(* CODESYS project aircomlib_v1_3_0.library
   Author: Piotr Kaźmierczuk
   Placeholder: AircomLibrary
   Title: AircomLibrary
   Version: 1.3.0
   Description: Biblioteka z używanymi na liniach produkcyjnych oraz maszynach testowych blokami funkcyjnymi, strukturami danych,wizualizacjami etc.
   Company: AirCom

Project tree, tasks and I/O mapping:
  libraries: Tc2_Math, * (Beckhoff Automation GmbH); Tc2_SerialCom, * (Beckhoff Automation GmbH); Tc2_Standard, * (Beckhoff Automation GmbH); Tc2_System, * (Beckhoff Automation GmbH); Tc2_Utilities, * (Beckhoff Automation GmbH); Tc3_Database, * (Beckhoff Automation GmbH); Tc3_EventLogger, * (Beckhoff Automation GmbH); Tc3_Module, * (Beckhoff Automation GmbH); Util, * (System); VisuDialogs, * (System); VisuSymbols, * (System)
  Common/
    2HandStart/
      BasicVer/
        function block fb2HandStartBasic [ST]
        data type st2HandStartBasic_InOuts
      function block fb2HandStart [ST]
      data type st2HandStart_InOuts
    Actuator/
      function block fbActuator [ST]: mClose, mOpen, mReset, mStop
      function block fbActuatorOOP [ST]: ACT_Stop, mClose, mOpen, mReset, mStop
      function block fbActuatorV2 [ST]: mClose, mOpen, mReset, mStop, Closed, CmdsCounter, Moving, Opened
      data type stActuatorDigInOut
      data type stActuatorInOuts
    AlarmTable/
      DUTs/
        data type enAlarmClasses
        data type stAlarmRowAppearanceData
        data type stAlarmTableRow
      function f_AlarmClassToUINT [ST]
      function f_AlarmEnableTest [ST]
      function block fbAlarmMasterTable [ST]: mPopRows, mPushRow, mReset
      function block fbAlarmSlaveTable [ST]: aMesagesPoped, mPushRow, mReset
    LoadCell/
      function fLoadCellCtrl [ST]
      function fLoadCellStatusToBOOL [ST]
      data type stLoadCell_InOutsData
    Maintenance/
      function block fbIIS_Restart [ST]
      function block fbTcAdsWcfHost_Restart [ST]
    Measurement_Analog/
      function fACRoundReal [ST]
      function block FB_FilterEx [ST]
      function block fbAnalogMeasurement [ST]
      function block fbAnalogMonitor [ST]
      function fMeanFilter [ST]
      function fMeasureStatusToBOOL [ST]
      function fRealValueFilter [ST]
      data type stMeasurementScalingData
    PulseCounter/
      function block fbPulseCounter [ST]
      function block fbPulseCounterPIM [ST]
    RecipeManager/
      DUTs/
        data type nRecipeManager_ErrorList
        data type stRecipeManager_ListEntry
      VISUs/
        visualisation vRecipeManager_Ctrl
        visualisation vRecipeManager_CtrlWide
      function block fbRecipeManager [ST]: ACT_DeleteRecipe, ACT_ReadRecipe, ACT_RefreshRecipeList, ACT_WriteRecipe
    SerialCom/
      function block fbSerialLinkCommunication [ST]
      data type stSerialComData
    String Functions/
      function block fbAcFormatString [ST]
      function block fbConcatStrings [ST]
      function fDataToHexStr [ST]
      function fGetStringUntil [ST]
      function fHexStrToData [ST]
      function fRemChar [ST]
    TimeProg/
      function block fbDateAndTimeCalc [ST]: mCalculate
      data type stAircomTimeStruct
    TimeTableStats/
      OOP_Version/
        function block fbTimeTable255 [ST]: mPushRow, mPushText, mReset, IsEmpty, IsFull, LastIndex
        interface I_TimeTable255: mPushRow, mPushText, mReset, IsEmpty, IsFull, LastIndex
        data type stTimeStatsRow255
      function block fbTimeTable [ST]: mPushRow, mPushText, mReset, IsEmpty, IsFull, LastIndex, MaxIndex
      interface I_TimeTable: mPushRow, mPushText, mReset, IsEmpty, IsFull, LastIndex, MaxIndex
      data type stTimeStatsRow
    function block fbBinaryFilter [ST]
    function block fbBlink [ST]
    function block fbLED_Blink [ST]
    function block fbOperationSynch [ST]
    function block fbPwmGenerator [ST]
    function block fbSequenceWork [ST]
    function block fbWriteStringToFile [ST]
  DataLoggers/
    function block fbTextDataLogger [ST]: mAddLine, mAppendCurrentLine, mEndLine, mIsActEmpty, mSaveBuffor
  DUTs/
    data type nBasicWorkStep
  PIM/
    DUTs/
      data type nPIM_ErrorCodes
      data type nPIM_EventClasses
      data type nPIM_MachineStates
      data type nPIM_ReportedNokSource
      data type nPIM_ReworkSelect
      data type stPIM_ExtDataRow
      data type stPIM_MachineParametersData
      data type stPIM_ServiceInOuts
      data type stPIM_StationSettings
      data type stPIM_StationStatus
    Interfaces/
      interface I_PIM: m_SqlInsertExtendedData, m_SqlSelLastOperationStatus, mGetStationData, mNewEvent, mNewServiceMessage, mSetNewMachineState, PartsCtr_NOK, PartsCtr_OK, prActiveErrorCode, prCMD, prCurrentMachineState, prErrorClassExt, prErrorConfirmActive, prExternalEvtWaitInQueue, prLastSavedStatus, prNokReportedSource, prOperEnded, prOperInProgress, prPimActive, prPimBlockWork, prPlcBlockWork, prReworkStatus, prStationDataOK, prTestMode, prUserLogged, prWorkPermission, prIsEol, prPartCodeNumber, prIsHidden, prLineName, prMachNumber, prStationAlias, prStationName
      interface I_SqlCmds: m_SqlInsAdditionalError, m_SqlInsCompressedAirConsumption, m_SqlInsDefectRelation, m_SqlInsEnergyConsumption, m_SqlInsertExtendedData, m_SqlSelInsStatus, m_SqlSelLastOperationStatus
      interface I_StationMachine: mGetParamsData
    POUs/
      function block fbPIM_Dummy [ST]: m_SqlInsertExtendedData, m_SqlSelLastOperationStatus, mGetStationData, mNewEvent, mNewServiceMessage, mSetNewMachineState
      function block fbPIM_MachineDummy [ST]: FB_init, mGetParamsData, mNewEvent
      function block fbPIM_SimplePimStation [ST]: PartsCtr_NOK, PartsCtr_OK, prActiveErrorCode, prCMD, prCurrentMachineState, prErrorClassExt, prErrorConfirmActive, prExternalEvtWaitInQueue, prLastSavedStatus, prNokReportedSource, prOperEnded, prOperInProgress, prPimActive, prPimBlockWork, prPlcBlockWork, prReworkStatus, prStationDataOK, prTestMode, prUserLogged, prWorkPermission, prIsEol, prPartCodeNumber, prIsHidden, prLineName, prMachNumber, prStationAlias, prStationName, m_SqlInsAdditionalError, m_SqlInsCompressedAirConsumption, m_SqlInsDefectRelation, m_SqlInsEnergyConsumption, m_SqlInsertExtendedData, m_SqlInsMachineParamsData, m_SqlSelInsStatus, m_SqlSelLastOperationStatus, m_SqlSelLineStationId, m_SqlSelMachineParamsCRC, m_SqlSelMachineParamsData, ACT_PimCmdsHandling, ACT_SqlDataReturnCmd, ACT_UpdatePimOutput, FB_init, mGetStationData, mNewEvent, mSendCmdToPIM
      function block fbPIM_Station_V3 [ST]: PartsCtr_NOK, PartsCtr_OK, prActiveErrorCode, prCMD, prCurrentMachineState, prErrorClassExt, prErrorConfirmActive, prExternalEvtWaitInQueue, prLastSavedStatus, prNokReportedSource, prOperEnded, prOperInProgress, prPimActive, prPimBlockWork, prPlcBlockWork, prReworkStatus, prStationDataOK, prTestMode, prUserLogged, prWorkPermission, prIsEol, prPartCodeNumber, prIsHidden, prLineName, prMachNumber, prStationAlias, prStationName, m_SqlInsAdditionalError, m_SqlInsCompressedAirConsumption, m_SqlInsDefectRelation, m_SqlInsEnergyConsumption, m_SqlInsertExtendedData, m_SqlInsMachineParamsData, m_SqlSelInsStatus, m_SqlSelLastOperationStatus, m_SqlSelLineStationId, m_SqlSelMachineParamsCRC, m_SqlSelMachineParamsData, ACT_PimCmdsHandling, ACT_SqlDataReturnCmd, ACT_UpdatePimOutput, FB_init, mGetStationData, mNewEvent, mNewEventCommon, mNewlnternalEvent, mNewServiceMessage, mSendCmdToPIM, mSetNewMachineState
      function block fbPIM_UserLogin [ST]: FB_init
      function fPIM_GetCmdPar [ST]
  ProdLineMachines/
    AssemblyPost/
      DUTs/
        data type nAssemblyPost_ErrorList
        data type stAssemblyPost_Settings
      VISUs/
        visualisation vAssemblyPost_Main
      function block fbAssemblyPost [ST]: FB_init, mGetParamsData, mNewEvent
    S02_ManometerTubeAssy/
      V1/
        DUTs/
          data type nManometerTubeAssy_ErrorCodes
          data type stManometerTubeAssy_InOuts
        function block fbManometerTubeAssy_V1 [ST]: FB_init, mGetParamsData, mNewEvent
      V2/
        DUTs/
          data type nManometerTubeAssy_V2_ErrorCodes
          data type stManometerTubeAssy_V2_InOuts
        function block fbManometerTubeAssy_V2 [ST]: FB_init, mGetParamsData, mNewEvent
    S05_BallsWheelPress/
      DUTs/
        data type nBallCounterPressPress_ErrorCodes
        data type stBallCounterWeightPress_InOuts
        data type stBallCounterWeightPress_Params
      function block fbBallCounterWeightPress [ST]: FB_init, mGetParamsData, mNewEvent
    S11_ResWelderTecna/
      DUTs/
        data type nTecnaResWelder_ErrorCodes
        data type stTecnaResWelder_InOuts
        data type stTecnaResWelder_TestParams
      function block fbTecnaResWelder [ST]: FB_init, mGetParamsData, mNewEvent
    S12_Hios/
      DUTs/
        data type nHIOS_ErrorList
        data type nHIOS_SerialCmds
        data type stHIOS_FastenExtData
        data type stHIOS_InOuts
        data type stHIOS_ScrewDriverParams
        data type stHIOS_TestParameters
      function block fbHIOS_ScrewDriver [ST]: ACT_SerialCom, FB_init, mGetParamsData, mNewEvent
    S13_FrontFanPress/
      DUTs/
        data type nFrontFanPress_ErrorCodes
        data type stFrontFanPress_InOuts
      function block fbFrontFanPress [ST]: FB_init, mGetParamsData, mNewEvent
    S18_ManometerCalib/
      DUTs/
        data type nManometerCalibration_ErrorCodes
        data type stManometerCalibration_InOuts
        data type stManometerCalibration_TestData
      function block fbManometerCalibration [ST]: FB_init, mGetParamsData, mNewEvent
    Sonictech/
      Fixtures/
        NoWeldLock/
          function block fbStFix_NoWeldLock [ST]
          data type nStFix_NoWeldLock_ErrorCodes
        S01_IndicatorAssembly/
          DUTs/
            data type nStFix_S01IndicatorAssy_ErrorCodes
            data type stStFix_S01IndicatorAssy_InOut
            data type stStFix_S01IndicatorAssy_Settings
          VISUs/
            SubFrame/
              visualisation vStFix_S01IndicatorAssy_SubDiag
              visualisation vStFix_S01IndicatorAssy_SubSettings
            visualisation vStFix_S01IndicatorAssy_Main
          function block fbStFix_S01IndicatorAssy [ST]
        S06_CarrierWheelLubrification/
          V1/
            DUTs/
              data type nStFix_S06CarrierAndWheelAssyGrease_ErrorCodes
              data type stStFix_S06CarrierAndWheelAssyGrease_InOuts
              data type stStFix_S06CarrierAndWheelAssyGrease_Settings
            function block fbStFix_S06CarrierAndWheelAssyGrease [ST]
          V2/
            DUTs/
              data type nStFix_S06CarrierAndWheelAssyGrease_V2_ErrorCodes
              data type stStFix_S06CarrierAndWheelAssyGrease_V2_InOuts
              data type stStFix_S06CarrierAndWheelAssyGrease_V2_Settings
            function block fbStFix_S06CarrierAndWheelAssyGrease_V2 [ST]
        S07_CarrierAssyWithPiston/
          V1/
            DUTs/
              data type nStFix_S07CarrierPistonAssy_ErrorCodes
              data type stStFix_S07CarrierPistonAssy_InOuts
              data type stStFix_S07CarrierPistonAssy_Settings
            function block fbStFix_S07CarrierPistonAssy [ST]
          V2/
            DUTs/
              data type nStFix_S07CarrierPistonAssy_V2_ErrorCodes
              data type stMachineSettingsHeatStamp
              data type stStFix_S07CarrierPistonAssy_V2_InOuts
              data type stStFix_S07CarrierPistonAssy_V2_Settings
            function block fbStFix_S07CarrierPistonAssy_V2 [ST]: ACT_HeatStamp, mNewEvent
        S08_CoolerClosure/
          V1/
            function block fbStFix_S08CoolerClosure [ST]
            data type nStFix_S08CoolerClosure_ErrorCodes
            data type stStFix_S08CoolerClosure_InOuts
          V2/
            DUTs/
              data type nStFix_S08CoolerClosure_V2_ErrorCodes
              data type stStFix_S08CoolerClosure_V2_InOuts
              data type stStFix_S08CoolerClosure_V2_Settings
            function block fbStFix_S08CoolerClosure_V2 [ST]
        S10_CoolerCarrierOrifice/
          function block fbStFix_S10CoolerCarrierOrifice [ST]
          data type stStFix_S10CoolerCarrierOrifice_InOuts
        S16_FixAndFrontFanDetection/
          DUTs/
            data type nStFix_S16PinWeldFfDetection_ErrorCodes
            data type stStFix_S16PinWeldFfDetection_InOuts
            data type stStFix_S16PinWeldFfDetection_Settings
          function block fbStFix_S16PinWeldFfDetection [ST]
        S17_EnclosurePressFix/
          DUTs/
            data type nStFix_S17EnclosureWelding_ErrorCodes
            data type stStFix_S17EnclosureWelding_InOuts
          function block fbStFix_S17EnclosureWelding [ST]
        function block fbStFixBaseTemplate [ST]: prFixError, prFixErrorID, prFixLocked, prFixReady, prFixReleased, prMachState, prTestMode, prTestOutputsActive, prUserLogged, prWeldingActive, actCheckForNewOrder, mAuxOper, mLock, mNewEvent, mRelease
        interface I_Fixture: prFixError, prFixErrorID, prFixLocked, prFixReady, prFixReleased, prMachState, prTestMode, prTestOutputsActive, prUserLogged, prWeldingActive, mAuxOper, mLock, mRelease
      SerialCom/
        DUTs/
          DataStruct/
            data type stSonicTech_SerialStructGenParamsRange
            data type stSonicTech_SerialStructProgParams
            data type stSonicTech_SerialStructSoftVer
            data type stSonicTech_SerialStructWeldParams
          data type nSonicTech_SerialCmdClasses
          data type nSonicTech_SerialCmdStatus
          data type nSonicTech_SerialCmdType
          data type stSonicTech_SerialCMD
        function block fbSonictechSerialCom [ST]: ACT_Test_Cmds, mAddToQueue, mFillSendBuffor
        function block fbSonictechSerialRcv [ST]
        interface I_SonicTech_SerialCom: mAddToQueue
      Welding Machine/
        DUTs/
          data type nSonicTech_ErrorList
          data type stSonicTech_DigInOuts
          data type stSonicTech_MachSettings
        VISUs/
          SubFrame/
            visualisation vSonictechUSWM_SubDiag
            visualisation vSonictechUSWM_SubSettings
            visualisation vSonictechUSWM_SubStatus
          visualisation vSonictechUSWM_Main
        function block fbSonictechUSWM [ST]: FB_init, mGetParamsData, mNewEvent, mNewMachEvent
  SQL/
    DUTs/
      DataSelectDUTs/
        data type stSQL_RetDataProdLineStat
        data type stSQL_RetDataProdMachParams
        data type stSQL_RetDataUserRole
      HMI_DUTs/
        data type stSQL_HMI_CoreNodesData
        data type stSQL_HMI_QueueData
      data type nSQL_CmdExecState
      data type nSQL_CmdTypes
      data type nSQL_ErrorCodes
      data type nSQL_UserRoles
      data type stSQL_ClientNode
      data type stSQL_SaveStatustParams
    VISUs/
      visualisation vSQL_Core_AlarmTab
      visualisation vSQL_CoreDiag
    function block fbSQL_Core [ST]: actConnectionCheck, IsCoreWork, m_ErrorAnalysis, mAddCmdToQueue, mPopCmdFromQueue
    function block fbSQL_CoreNode [ST]: ACT_Init, mSaveError
    interface I_SQL_Core: IsCoreWork, mAddCmdToQueue
  VisionSensors/
    Balluff BVS/
      function block fbBvsControl [ST]: mNewInspection, mReadInspectionId, mSetInspectionId
      function block fbBvsControl_ComIO [ST]: mNewInspection, mReadInspectionId, mSetInspectionId
      data type stBVS_DigInOut
    Cognex/
      function block fbCognexIS280Control [ST]: mNewInspection, mReadInspectionId, mSetInspectionId
      data type stCognexIS280_DigInOut
    Keyence/
      IV3/
        data type stKeyenceIV3_DigInOut
      function block fbKeyenceIVControl [ST]: mNewInspection, mReadInspectionId, mSetInspectionId
      function block fbKeyenceIVControl_ComIO [ST]: mNewInspection, mReadInspectionId, mSetInspectionId
      data type stKeyence_DigInOut
    interface I_VisionSensorSTD: mNewInspection, mReadInspectionId, mSetInspectionId
    data type stVisionSensor_DigInOut
  text list GlobalTextList
  global variables GVL_Aircom
  program ReadMe [ST]
*)

// Common/2HandStart/BasicVer/st2HandStartBasic_InOuts
TYPE st2HandStartBasic_InOuts :
STRUCT
	bEmergButton_NC 	AT %I* :BOOL;		// TRUE- Emergency button released (inactive) , FALSE- Pressed (safety function activated)
	bLeftStart_NC 		AT %I* :BOOL;		// First button - NC contact
	bRightStart_NO 		AT %I* :BOOL;		// Second button - NO contact
END_STRUCT
END_TYPE

// Common/2HandStart/st2HandStart_InOuts
TYPE st2HandStart_InOuts :
STRUCT
	bSafetyStatus_NC 	AT %I* :BOOL;		// 1- gdy układ nie uzbrojony i sprawny (zezwolenie na reset), 0- gdy uzbrojony lub uszkodzony
	bEmergButton_NO 	AT %I* :BOOL;		// 1- Stop bezpieczeństwa wciśnięty, 0- zwolniony
	bLeftStart_NC 		AT %I* :BOOL;
	bRightStart_NO 		AT %I* :BOOL;
	bLeftStart_NO 		AT %I* :BOOL;
	bRightStart_NC 		AT %I* :BOOL;
	bSafetyReset 		AT %Q* :BOOL;		// Uzbrojenie układu bezpieczeństwa
END_STRUCT
END_TYPE

// Common/Actuator/stActuatorDigInOut
TYPE stActuatorDigInOut :
STRUCT
	bI_Opened AT %I*:BOOL;							// Sygnał z krańcówki otwarcia
	bI_Closed AT %I*:BOOL;							// Sygnał z krańcówki zamknięcia
	bQ_Open AT %Q*:BOOL:= FALSE;					// Sygnał do zaworu otwierania (w przypadku zaworu jednocewkowego podłączyć tylko to wyjście)
	bQ_Close AT %Q*:BOOL:= FALSE;					// Sygnał do zaworu zamykania
END_STRUCT
END_TYPE

// Common/Actuator/stActuatorInOuts
TYPE stActuatorInOuts :
STRUCT
	bI_Opened AT %I*:BOOL;							// Sygnał z krańcówki otwarcia
	bI_Closed AT %I*:BOOL;							// Sygnał z krańcówki zamknięcia
	bQ_Open AT %Q*:BOOL:= FALSE;					// Sygnał do zaworu otwierania (w przypadku zaworu jednocewkowego podłączyć tylko to wyjście)
	bQ_Close AT %Q*:BOOL:= FALSE;					// Sygnał do zaworu zamykania
END_STRUCT
END_TYPE

// Common/AlarmTable/DUTs/enAlarmClasses
{attribute 'qualified_only'}
{attribute 'strict'}
{attribute 'to_string'}
TYPE enAlarmClasses :
(
	// Lista klas alarmów - identyfikatory nie powinny zmieniać wartości
	None := 0,					// Logowanie wyłączone
	Info := 1,					// Logowanie podstawowych informacji
	Warning := 2,				// Ostrzeżenia
	Error := 4,	
	Quality := 8,
	Maintenance := 16,
	IT := 32,
	Developer := 64);
END_TYPE

// Common/AlarmTable/DUTs/stAlarmRowAppearanceData
TYPE stAlarmRowAppearanceData :
STRUCT
	sFontName:STRING:= 'Arial';
	iFontSize:INT:= 10;			// Rozmiar czcionki
	dwFontFlags:DWORD; 			// Flagi 1-italic, 2-bold, 4-underlined, 8-deleted, można je sumować
	dwTextColor:DWORD:=16#FF404040;			// Format koloru - 16#TTRRGGBB;
	dwAlignmentFlags:DWORD;		// Wyrównanie tekstu 0-TopLeft, 1-CenterHor, 2-Right, 4-CenterVert, 8-below
	dwBackgroundColor:DWORD:=16#FFCDCDCD;	// Kolor tła
	dwFrameColor:DWORD:=16#FF585858;		// Kolor ramki
	iFrameWidth:INT:= 1;					// Rozmiar ramki
END_STRUCT
END_TYPE

// Common/AlarmTable/DUTs/stAlarmTableRow
TYPE stAlarmTableRow :
STRUCT
	dtEventTime:DT;
	sMachineId:STRING(30);
	sEventDescription:STRING;
	dwErrorCode:DWORD;
	uiRepeatQty:UINT := 0;
	nAlarmClass:enAlarmClasses;
END_STRUCT
END_TYPE

// Common/LoadCell/stLoadCell_InOutsData
TYPE stLoadCell_InOutsData :
STRUCT
	wStatus		AT %I* : WORD;	// .1-Overrange, .3-Data invalid, .6-Error, .7-Calib in progress, .9-Steady state, .13-SyncErr, .15-TxPDO_Toggle
	rValue		AT %I* : REAL;	// Wartość siły w [N]
	wControl	AT %Q* : WORD;	// .0-Start calibration, .1-Disable calib., .2-InputFreeze, .4-Tara
END_STRUCT
END_TYPE

// Common/Measurement_Analog/stMeasurementScalingData
TYPE stMeasurementScalingData :
STRUCT
	rScalingRawValue_I:REAL := 0;	// Wartość surowa pomiaru w I punkcie pomiarowym
	rScalingEngValue_I:REAL	:= 0;		// Wartość inżynierska pomiaru w I punkcie pomiarowym
	rScalingRawValue_II:REAL := 32767;	// Wartość surowa pomiaru w II punkcie pomiarowym
	rScalingEngValue_II:REAL := 10;	// Wartość inżynierska pomiaru w II punkcie pomiarowym
END_STRUCT
END_TYPE

// Common/RecipeManager/DUTs/nRecipeManager_ErrorList
{attribute 'qualified_only'}
{attribute 'strict'}
{attribute 'to_string'}
TYPE nRecipeManager_ErrorList :
(
	NoError := 0,
	ReloadRecipeListError:= 1,
	WriteRecipeError := 2,
	ReadRecipeError := 3,
	WriteSizeError:= 4,
	ReadSizeError:= 5,
	StructToBig:= 6,
	FileOpenError:= 7,
	FileCloseError:= 8,
	ReadRecipeTimeout:= 9,
	WriteRecipeTimeout:= 10,
	BadCRC:= 11,
	CommandStartProgramError:=12,
	FileDeleteError:=13,
	DeleteRecipeTimeout := 14
);
END_TYPE

// Common/RecipeManager/DUTs/stRecipeManager_ListEntry
TYPE stRecipeManager_ListEntry :
STRUCT
	sFileName:STRING;
	dtCreationTime:DT;
END_STRUCT
END_TYPE

// Common/SerialCom/stSerialComData
TYPE stSerialComData :
STRUCT
	fbSerialCom			: fbSerialLinkCommunication;	// Blok odpowiedzialny za komunikacjię
	RxBufferEL			: ComBuffer;	// Receive data buffer; used with all receive function blocks *)
	TxBufferEL			: ComBuffer;	// Transmit data buffer; used with all receive function blocks 
END_STRUCT
END_TYPE

// Common/TimeProg/stAircomTimeStruct
TYPE stAircomTimeStruct :
STRUCT
	bTimeValid		: BOOL;					// Jeśli true dane w strukturze są aktualne
	stTimeStruct 	: TIMESTRUCT;			// Struktura z danymi rokiem, miesiącem, dniem itp w formacie WORD
	dtActualDate 	: DT;					// Aktualny czas typ DT
	tCycleTime		: TIME;					// Czas cyklu sterownika PLC
	tActualTime		: TIME;					// Aktualny czas
	sTimeString		: STRING(19);			// String z aktualną datą w formacie : YYYY-MM-DD hh:mm:ss
	sLogTimeString		: STRING(18);			// String z aktualną datą w formacie : MM-DD hh:mm:ss.uuu
	diPLC_UpTimeSeconds	: DINT:= 0;			// Licznik czasu pracy PLC w sekundach
	dtPLC_UpTime	: DT;					// Czas w którym PLC wystartował					
	// Znaczniki nowych okresów czasu
	bNew_Second_IMP, bNew_Minute_IMP, bNew_Hour_IMP, bNew_Day_IMP, bNew_Week_IMP, bNew_Month_IMP, bNew_Year_IMP:BOOL;	// Impuls nowej sekundy, minuty, godziny, dnia, tygodnia, miesiąca, roku
	// Znaczniki zmian
	bNew_Shift		: BOOL;					// Znacznik nowej zmiany (impuls)
	wWeekNb			: WORD;					// Numer tygodnia
	uiShiftNumber	: UINT;					// Numer aktualnej zmiany 1, 2 lub 3
END_STRUCT
END_TYPE

// Common/TimeTableStats/OOP_Version/stTimeStatsRow255
{attribute 'enable_dynamic_creation'}
TYPE stTimeStatsRow255 :
STRUCT
	sStepName:STRING(255);
	rStepTime:REAL;
END_STRUCT
END_TYPE

// Common/TimeTableStats/stTimeStatsRow
TYPE stTimeStatsRow :
STRUCT
	sStepName:STRING;
	rStepTime:REAL;
END_STRUCT
END_TYPE

// DUTs/nBasicWorkStep
{attribute 'qualified_only'}
{attribute 'strict'}
TYPE nBasicWorkStep :
(
	StartUpInicialization	 	:= 0,
	Inicialization			 	:= 5,
	WaitForStart	 			:=10,
	LockStation 				:=90,
	WaitForConfirm				:=94,
	ConfirmInProgress			:=95
);
END_TYPE

// PIM/DUTs/nPIM_ErrorCodes
{attribute 'qualified_only'}
{attribute 'strict'}
TYPE nPIM_ErrorCodes :
(
	// Common errors	
	NoError := 0,										// Brak błędu
	UnKnownAlarm := 53,									// Niezidentyfikowany alarm maszyny
	UnKnownLock := 54,									// Niezidentyfikowana blokada maszyny
	MachErrorWhenNoErrorCode := 56,						// Maszyna w oczekiwaniu na reset, ale brak błędu
	ProgramError := 90,									// Błąd w konfiguracji oprogramowania - zerowy wskaźńik itp
	SelectStationIdError := 230,						// Błąd pobrania ID stacji z bazy danych
	StatusSaveError := 89,								// Błąd zapisu statusu
	InputDependencyError := 99,							// Błąd zależności wejściowych (brak referencji)
	ResetTimeout := 518,								// Timeout resetu maszyny
	NoConfiguredOutPart := 150, 						// Brak skonfigurowanej części wyjściowej dla stanowiska
	NoMatchingParamsForComponent := 151,				// Brak zdefiniowanych parametrów dla komponentu
	ParamsMismatchPLCandDB := 152,						// Rozbieżność parametrów w PLC i w DB
	NoDbConnWorkAllowedTemporary := 153,				// Brak połączenia do DB, stacja dopuszczona warunkowo
	ParamsSaveToDB_Error := 154,						// Błąd wysłania parametrów programu do bazy danych
	ParamsReadFromDB_Error := 155,						// Błąd pobierania parametrów programu z bazy danych
	MachineParametersNoUpdated := 156					// Błąd odświeżenia danych z maszyny
);
END_TYPE

// PIM/DUTs/nPIM_EventClasses
{attribute 'qualified_only'}
{attribute 'to_string'}
{attribute 'strict'}
TYPE nPIM_EventClasses :
(
	NoError := 0,				// Brak błędu/alarmuwiadomości
	Message := 1,				// Wiadomość do użytkownika - baner wyświetlony przez x sekund lub do startu nowej operacji 
	AlarmAutoConfirm := 2,		// Alarm stanowiska który działa tak jak wprzypadku zwykłego alarmu ale zostaje automatycznie potwierdzony przy starcie nowej operacji 
	Alarm := 3,					// Alarm stanowiska - błąd związany z pracą maszyny, potwierdzenie nie wymaga lidera, nie ma pytania o rework
	Error := 4					// Blokowanie stanowiska powiązane z częścią - zawsze błąd potwierdza lider, sprawdzeny jest zapis statusu oraz część jest blokowana w kowadle (+ pytanie o rework)
);
END_TYPE

// PIM/DUTs/nPIM_MachineStates
{attribute 'qualified_only'}
{attribute 'strict'}
{attribute 'to_string'}
(*	Na podstawie stanu/kroków maszyny wydawane jest zezwolenie na przejście do danego kroku (zezwolenie na pracę, reset błędu itp) oraz zapisywany jest status operacji. 
	Wzorzec postępowania
	1. _2_ReadyForNewOperation - maszyna gotowa do wykonania operacji,
	2. _3_NewOperationStarted - gdy maszyna wystartowała blok stacji zapamiętuje konieczność zapisu statusu, 
	3. _5_OperationEndedOK lub _7_ErrorOccurr - informacja jaki status trzeba zapisać
	Jeśli po starcie operacji był sygnał _9_ErrorOccurr a nie było zapisu statusu (zgłoszenie błędu) i jest stan _10_WaitForReset to zapis statusu przez stację PIM

	Reset błędów: Blok maszyny czeka w stanie _8_WaitForReset zezwolenie na przejście do kolejnego kroku (_9_ResetInProgress). Jeśli reset zakończony powodzeniem zawsze kończy się stanem
	_0_Standby_NotReady (przy tym przejściu resetowane są zmienne od alarmów jeśli był aktywny błąd zewnętrzny)
*)
TYPE nPIM_MachineStates :
(
	_0_Initialization	 		:= 100,	// Inicjalizacja maszyny
	_0_Standby_NotReady 		:= 0,	// Maszyna w oczekiwaniu na stan gotowości
	_1_InManualControl		 	:= 1,	// Maszyna w sterowaniu serwisowym/ręcznym 
	_2_ReadyForNewOperation 	:= 2,	// Maszyna gotowa na wykonanie kolejnej operacji ( sygnał nie uwzględnia zezwolenia na pracę
	_3_NewOperationStarted 		:= 3,	// Nowa operacja rozpoczęta - jest zezwolenie, przygotowanie kowadła
	_4_OperationInProgress 		:= 4,	// Operacja w trakcie
	_5_OperationEndedOK			:= 5,	// Operacja zakończona ze statusem OK
	_6_ReturningToBaseState		:= 6,	// Powrót do stanu początkowego po zezwoleniu przez PIM
	_7_ErrorOccurr				:= 7,	// Wystąpił błąd - blokowanie części ustawianie maszyny w odpowiednim stanie	
	_8_WaitForReset				:= 8,	// Oczekiwanie na sygnał reset
	_9_ResetInProgress			:= 9	// Trwa reset maszyny
);
END_TYPE

// PIM/DUTs/nPIM_ReportedNokSource
{attribute 'qualified_only'}
{attribute 'strict'}
TYPE nPIM_ReportedNokSource :
(
	none := 0,
	FromPrevStation := 1,
	FromMach := 2,
	FromBox := 3,
	Error_UnknownSource := 4
);
END_TYPE

// PIM/DUTs/nPIM_ReworkSelect
{attribute 'qualified_only'}
{attribute 'strict'}
TYPE nPIM_ReworkSelect :
(
	none := 0,
	yes := 1,
	no := 2
);
END_TYPE

// PIM/DUTs/stPIM_ExtDataRow
TYPE stPIM_ExtDataRow :
STRUCT
	sName:STRING(63);		// Nazwa parametru
	sValue:STRING(31);		// Wartość parametru
END_STRUCT
END_TYPE

// PIM/DUTs/stPIM_MachineParametersData
TYPE stPIM_MachineParametersData :
STRUCT
	abMachineParameters: ARRAY [1..1000] OF BYTE;		// Wskaźnik do parametrów pracy maszyny
	uiMachineParametersSize: UINT;						// Rozmiar struktury parametrów pracy maszyny
	wActualCRC16SumInMachine: WORD;						// Aktualna suma CRC16 obliczona z parametrów
END_STRUCT
END_TYPE

// PIM/DUTs/stPIM_ServiceInOuts
(*
	Lista zmiennych które są wymieniane pomiędzy PLC a PIM, nazewnictwo zmiennych poszukiwanych w programie MAIN:
		stStacjaXXXX	- gdzie XXXX to nazwa stanowiska w PIM np. stStacjaLJ01, stStacjaLL19 - dla stanowisk z pojedynczą maszyną...
		stStacjaXXXX_MY	- gdzie XXXX to jw. nazwa stanowiska, Y to numer maszyny na stanowisku np. stStacjaLJ05_M1, stStacjaLJ05_M2 - dla stanowisk wielomaszynowych
	Update 01.03.2024r. - nowe nazwy zmiennych
		stStation_L{nazwa linii}_S{nazwa stanowiska}[_M{numer maszyny}] - rzeczy w klamrach {} zastępujemy zgodnie ze stanowiskiem, parametr z numerem maszyny w nawiasach [] jest konieczny tylko gdy maszyn jest >1
*)
TYPE stPIM_ServiceInOuts :
STRUCT
	//Dane in/out systemu PIM
	bPIMActive : BOOL := TRUE;					// jeśli TRUE system PIM wlaczony
	bUserLogged : BOOL := FALSE; 				// z PIM blokowanie stanowiska gdy nikt nie jest zalogowany - 1 nie zalogowany, 0 - zalogowany  
	bWorkBlock_PIM : BOOL;						// z PIM blokowane - 1 blokada, 0 praca
	bWorkBlock_PLC : BOOL;						// z PLC, jesli TRUE stanowisko pozostaje zablokowane z powodu błędu z operacją, trzeba wysłać status części NOK do bazy danych z kodem błędu
	bAlarmPLC : BOOL;							// z PLC, jesli TRUE stanowisko pozostaje zablokowane z powodu błędu maszyny, brak zapisu statusu (można zapisać dodatkowy kod błędu)
	bNonBlockingAlarm : BOOL;					// do użytku w kodzie PLC - gdy true i jest aktywny AlarmStanowiska, stanowisko nie jest blokowane (jedynie wyświetlany jest alarm - potwierdzenie po starcie nowej operacj, zniknięciu powodu błędu)
	bConfirmEvent : BOOL;						// z PIM potwierdzenie bledu, komunikatu przez operatora
	bTestMode : BOOL;							// jesli TRUE stacja nie sprawdza poprzedniej operacji 
	sErrorCodePLC : STRING(255); 				// komunikat o bledzie dzialania maszyny np kontaktron, e-stop
	sPlcServiceMessage : STRING(255);			// Komunikat do PIM wyświetlany na dolnym pasku
	sStatusNokAndErrorID : STRING(255);			// Informacja odczytywana przez PIM aby zapisać relację błędów - postaci {IdStatusu}:{IdBłędu}
	sCmdPIM2PLC:STRING(255);					// Komunikaty wysyłane z PIM do PLC (np. informacja o nowym boxie, zgłoszeniu części NOK itp)
	sCmdPLC2PIM:STRING(255);					// Komunikaty wysyłane z PLC do PIM  (np. zapytanie o licznik części itp.)
END_STRUCT
END_TYPE

// PIM/DUTs/stPIM_StationSettings
TYPE stPIM_StationSettings :
STRUCT
	bCheckMachineSettings:BOOL := FALSE;			// Sprawdzaj parametry maszyny
	bAutoRetooling:BOOL;							// Jeśli nastąpiło przezbrojenie automatycznie pobierz nowe parametry z bazy danych (o ile istnieją)
	bSkipCheckStatusSaveResult:BOOL:= FALSE;		// Czekaj z gotowością do nowej operacji aż status zostanie poprawnie zapisany
END_STRUCT
END_TYPE

// PIM/DUTs/stPIM_StationStatus
TYPE stPIM_StationStatus :
STRUCT
	// Dane informacyjne z bloczka obsługi PIM
	sLine				: STRING(31);	// Nazwa linii
	sStation			: STRING(31);	// Nazwa stacji
	sNazwaStanowiska 	: STRING(16);	// Id stanowiska (stanowisko + nr maszyny)
	
	stStationSqlData:stSQL_RetDataProdLineStat;	// Dane stanowiska - Id, AutSaveErrors itp	
	iMachineNumber 		: INT;			// Numer maszyny na stanowisku
	bIsHidden 			: BOOL;			// Czy ukrywanie zapisu statusu
	
			
(*	// Liczniki części oraz błędów
	iOutBoxQty, iOutBoxTargetQty: INT;			// liczba ilość części w pudełku wyjściowym - zmienne inkrementowane/dekrementowane tylko w bloczku PIM! Uaktualniane w FB maszyny tylko jeśli był restart sterownika.
	iPartsOK:INT;								// Licznik części OK wyprodukowanych na aktualnej zmianie
	iPartsNOK:INT;								// Licznik części NOK wyprodukowanych na aktualnej zmianie
	iPartsNotSaved:INT;							// Licznik błędnych statusów OK/NOK na aktualnej zmianie
	rEnergyConsumption:REAL;					// Zużycie energii na stanowisku	
	*)
END_STRUCT
END_TYPE

// ProdLineMachines/AssemblyPost/DUTs/nAssemblyPost_ErrorList
{attribute 'qualified_only'}
{attribute 'strict'}
TYPE nAssemblyPost_ErrorList :
(
	NoError := 0,
	PartRemovedToFast := 93,				// Złożenie zbyt szybko usunięte z kowadła
	PartInsertedToFast := 94,				// Złożenie zbyt szybko umieszczone w kowadle po usunięciu starego
	InputDependencyError := 99
);
END_TYPE

// ProdLineMachines/AssemblyPost/DUTs/stAssemblyPost_Settings
TYPE stAssemblyPost_Settings :
STRUCT
	bMonitorON_Time:BOOL;
	bMonitorOFF_Time:BOOL;
	rRequiredTimeON:REAL;
	rRequiredTimeOFF:REAL;
END_STRUCT
END_TYPE

// ProdLineMachines/S02_ManometerTubeAssy/V1/DUTs/nManometerTubeAssy_ErrorCodes
{attribute 'qualified_only'}
{attribute 'strict'}
{attribute 'to_string'}
TYPE nManometerTubeAssy_ErrorCodes :
(
	// Błędy ogólne
	NoError := 0,
	UnKnownAlarm := 53,						// Niezidentyfikowany alarm maszyny
	UnKnownLock := 54,						// Niezidentyfikowana blokada maszyny
	ProgramConfigError := 90,				// Błąd w konfiguracji programu
	ResetTimeout := 518,					// Timeout resetu maszyny
	SafetySystemNotArmed := 614,			// System safety nie uzbrojony
	NoMachineReactionOnStartSig := 140,		// Brak reakcji na sygnał startu (brak wysunięcia siłownika - brak powietrza itp.)
	TwoHandStartReleasedToEarly := 96,		// Dwustart zwolniony zbyt wcześnie
	
	TwoHandStartContactsError := 130,		// Błąd styków dwustartu
	WorkPosAchieveTimeout := 131,			// Nie osiągnięto pozycji roboczej w zadanym czasie
	OperInteruptedBeforeWorkPos := 132,		// Za wcześnie puszczono dwustart - część nie wprasowana
	WorkPosLost := 138,						// Utracona pozycja robocza (możliwy brak części)
	HomePosAchieveTimeout := 139			// Nie osiągnięto pozycji bazowej w zadanym czasie
//	InConsistentSignalsFromSensors := 1000	// Niewłaściwe odczyty stanów z czujników - ingerencja zewnętrzna 
);
END_TYPE

// ProdLineMachines/S02_ManometerTubeAssy/V1/DUTs/stManometerTubeAssy_InOuts
TYPE stManometerTubeAssy_InOuts :
STRUCT
	st2HandStartIO			: st2HandStartBasic_InOuts;	// Sygnały z układu dwu-startu
	bHandleWorkPos			AT %I*: BOOL;	
	bHandleHomePosV2		AT %I*: BOOL;	// USed only with V2 wersion
	bPressWorkPos			AT %I*: BOOL;	
	bPressHomePos			AT %I*: BOOL;	
	bPressValve_Q			AT %Q*: BOOL;	
END_STRUCT
END_TYPE

// ProdLineMachines/S02_ManometerTubeAssy/V2/DUTs/nManometerTubeAssy_V2_ErrorCodes
{attribute 'qualified_only'}
{attribute 'strict'}
{attribute 'to_string'}
TYPE nManometerTubeAssy_V2_ErrorCodes :
(
	// Błędy ogólne
	NoError := 0,
	UnKnownAlarm := 53,						// Niezidentyfikowany alarm maszyny
	UnKnownLock := 54,						// Niezidentyfikowana blokada maszyny
	ProgramConfigError := 90,				// Błąd w konfiguracji programu
	ResetTimeout := 518,					// Timeout resetu maszyny
	SafetySystemNotArmed := 614,			// System safety nie uzbrojony
	NoMachineReactionOnStartSig := 140,		// Brak reakcji na sygnał startu (brak wysunięcia siłownika - brak powietrza itp.)
	NoWorkPermittionFromPIM := 84,			// Brak zezwolenia na pracę
	TwoHandStartReleasedToEarly := 96,		// Dwustart zwolniony zbyt wcześnie
	PusherHomePositionError:= 120,			//Praska nie w pozycji bazowej
	PusherWorkPositionError:= 121,			//Praska nie w pozycji pracy
	CartridgeHomePositionError:= 122,		//Wózeczek nie w pozycji bazowej
	CartridgeWorkPositionError:= 123,		//Wózeczek nie w pozycji pracy
	WorkPosAchieveTimeout := 131,			// Nie osiągnięto pozycji roboczej w zadanym czasie
	OperInteruptedBeforeWorkPos := 132,		// Za wcześnie puszczono dwustart - część nie wprasowana
	WorkPosLost := 138,						// Utracona pozycja robocza (możliwy brak części)
	HomePosAchieveTimeout := 139,			// Nie osiągnięto pozycji bazowej w zadanym czasie
	OperationTooEarly	:= 182				// Operacja została wykonanna w zbyt krótkim czasie 
);
END_TYPE

// ProdLineMachines/S02_ManometerTubeAssy/V2/DUTs/stManometerTubeAssy_V2_InOuts
TYPE stManometerTubeAssy_V2_InOuts :
STRUCT
	st2HandStartIO			: st2HandStartBasic_InOuts;	// Sygnały z układu dwu-startu
	bMoverWorkPos			AT %I*: BOOL;	
	bPressWorkPos			AT %I*: BOOL;	
	bPressHomePos			AT %I*: BOOL;	
	bMoveValve_Q			AT %Q*: BOOL;
	bPressValve_Q			AT %Q*: BOOL;	
END_STRUCT
END_TYPE

// ProdLineMachines/S05_BallsWheelPress/DUTs/nBallCounterPressPress_ErrorCodes
{attribute 'qualified_only'}
{attribute 'strict'}
{attribute 'to_string'}
TYPE nBallCounterPressPress_ErrorCodes :
(
		// Błędy ogólne
	NoError := 0,
	UnKnownAlarm := 53,						// Niezidentyfikowany alarm maszyny
	UnKnownLock := 54,						// Niezidentyfikowana blokada maszyny
	ProgramConfigError := 90,				// Błąd w konfiguracji programu
	ResetTimeout := 518,					// Timeout resetu maszyny
	SafetySystemNotArmed := 614,			// System safety nie uzbrojony
	NoMachineReactionOnStartSig := 140,		// Brak reakcji na sygnał startu (brak wysunięcia siłownika - brak powietrza itp.)
	TwoHandStartReleasedToEarly := 96,		// Dwustart zwolniony zbyt wcześnie

	WorkPosAchieveTimeout := 131,			// Nie osiągnięto pozycji roboczej w zadanym czasie
	OperInteruptedBeforeWorkPos := 132,		// Za wcześnie puszczono dwustart - część nie wprasowana
	WorkPosLost := 138,						// Utracona pozycja robocza (możliwy brak części)
	HomePosAchieveTimeout := 139,			// Nie osiągnięto pozycji bazowej prasy w zadanym czasie
	BallsNotPresentAfterPushing := 142

);
END_TYPE

// ProdLineMachines/S05_BallsWheelPress/DUTs/stBallCounterWeightPress_InOuts
TYPE stBallCounterWeightPress_InOuts :
STRUCT
	bPressUpPosition		AT %I* :BOOL;
	bPressDownPosition		AT %I* :BOOL;
	bBallSensorInWheel 		AT %I* :ARRAY [1..3] OF BOOL;
	bWheelPresenceSensor 	AT %I* :BOOL;
	bBallsInContainer		AT %I* :BOOL;
	bWibrationFeederStatus	AT %I* :BOOL;
	bPressValve_Q			AT %Q* :BOOL;		//
	bWibrationFeeder_Q		AT %Q* :BOOL;		//
END_STRUCT
END_TYPE

// ProdLineMachines/S05_BallsWheelPress/DUTs/stBallCounterWeightPress_Params
 TYPE stBallCounterWeightPress_Params :
STRUCT
	bBallsCheck			: BOOL := TRUE;
	iEnFeederEveryNCycles	: INT := 30;
	rFeederOnTime_S			: REAL := 60.0;	
END_STRUCT
END_TYPE

// ProdLineMachines/S11_ResWelderTecna/DUTs/nTecnaResWelder_ErrorCodes
{attribute 'qualified_only'}
{attribute 'strict'}
{attribute 'to_string'}
TYPE nTecnaResWelder_ErrorCodes :
(
		// Błędy ogólne
	NoError 						:= 0,
	ProgramConfigError 				:= 90,				// Błąd w konfiguracji programu
	SensorWorkError					:= 183,
	NoPartDetected 					:= 190,
	InvalidWeldOrder_FirstLeft		:= 192
);
END_TYPE

// ProdLineMachines/S11_ResWelderTecna/DUTs/stTecnaResWelder_InOuts
TYPE stTecnaResWelder_InOuts :
STRUCT
	stSerialCom					: stSerialComData;
	bLeftMotorSensor			AT %I*: BOOL;	
	bRightMotorSensor			AT %I*: BOOL;	
	bEndCycle					AT %I*: BOOL;	
	bWorkPermission_Q			AT %Q*: BOOL;	
	bProgramChange				AT %Q*: BOOL; //Wyjście pozalające na przestawienie programu na zgrzewarce TECNA 
END_STRUCT
END_TYPE

// ProdLineMachines/S11_ResWelderTecna/DUTs/stTecnaResWelder_TestParams
TYPE stTecnaResWelder_TestParams :
STRUCT
	bReworkMode_EN				: BOOL;			// Tryb reworku - gdy włączony konektor lewy zgrzewa się innym programem niż prawy (przełaczanie programów aktywne)
	bCheckWeldsOrder			: BOOL;			// Jeśli włączone Tecna sprawdza, czy pierwszy zgrzew nastąpił z lewej strony, następnie z prawej. Nie odwrotnie!
	bResetWhenNokReported		: BOOL;			// Gdy operator zgłosi NOK z maszyny cykl pracy jest resetowany do stanu początkowego
END_STRUCT
END_TYPE

// ProdLineMachines/S12_Hios/DUTs/nHIOS_ErrorList
{attribute 'qualified_only'}
{attribute 'strict'}
{attribute 'to_string'}
TYPE nHIOS_ErrorList :
(
	// Błędy ogólne
	NoError := 0,
	UnKnownAlarm := 53,						// Niezidentyfikowany alarm maszyny
	UnKnownLock := 54,						// Niezidentyfikowana blokada maszyny
	SelectStationIdError := 230,			// Brak pobranego Id stacji
	StatusSaveError := 89,					// Błąd zapisu statusu
	ResetTimeout := 518,					// Timeout resetu maszyny
	ProgramConfigError := 90,				// Błąd w konfiguracji programu
	SafetySystemNotArmed := 614,			// System safety nie uzbrojony
	NoMachineReactionOnStartSig := 140,		// Brak reakcji na sygnał startu (brak wysunięcia siłownika - brak powietrza itp.)

	MotorPulledFromFixWhenLocked := 273,	// Silnik usunięty z uchwytu gdy był zablokowany
	OverMilion_ResetReq	:= 2,	
	Rcv_Bad_CRC 		:= 60,
	RcvBadInputParams 	:= 61,
	RcvByteBlockError 	:= 62,
	RcvTimeout 			:= 63,
	RcvBadSuffix 		:= 64,
	RcvBufferOverflow 	:= 65

);
END_TYPE

// ProdLineMachines/S12_Hios/DUTs/nHIOS_SerialCmds
{attribute 'qualified_only'}
{attribute 'strict'}
TYPE nHIOS_SerialCmds :
(
	NoCommand := 0,					// Bezczynność
	AskForWorkParams := 1,			// Zapytanie o parametry
	AskForStartUpNb := 2,			// Zapytanie o ilosc zalaczen wkretaka
	AskForScrewdriverType := 3,		// Zapytanie o typ wkretaka
	ErrorReset := 4,				// Reset bledu
	ResetScrewsCounter := 5,		// Reset licznika śrub do wkręcenia
	LockScrewDriver := 6,			// Zablokowanie wkretaka
	UnLockScrewDriver := 7			// Odblokowanie wkretaka
);
END_TYPE

// ProdLineMachines/S12_Hios/DUTs/stHIOS_FastenExtData
TYPE stHIOS_FastenExtData :
STRUCT
	i1ScrewPulses:INT;
	i2ScrewPulses:INT;
END_STRUCT
END_TYPE

// ProdLineMachines/S12_Hios/DUTs/stHIOS_InOuts
TYPE stHIOS_InOuts :
STRUCT
	stSerialCom					: stSerialComData;
	bPartReleaseSignal	AT %I*	: BOOL;	
	bMotorSensor		AT %I*	: BOOL;	
	bMotorLockValve_Q	AT %Q*	: BOOL;		
END_STRUCT
END_TYPE

// ProdLineMachines/S12_Hios/DUTs/stHIOS_ScrewDriverParams
TYPE stHIOS_ScrewDriverParams :
STRUCT
	iSystemConstAR:INT;			// Współczynnik uczenia 0/5/10/15/20%
	iScrewsToFastenAn:INT;		// Liczba śrub do wkręcenia
	iMinPulseAc:INT;			// Minimalna liczba impulsów PASS
	iMaxPulseAC:INT;			// Maksymalna liczba impulsów PASS
	iBuzzerScrewsDoneTimeAt:INT;	// Długość sygnału dziwiękowego po wkręceniu wszystkich śrub
	iCntTimeForReverseOperationAr:INT;	// Czas operacji w przypadku cofania???
	iSystemSettingAd:INT;			//Konfiguracja systemu buzzer / reverse counting
	iErrorTypesDetectionAU:INT;		// Typ detekcji błędu - monitorowanie ograniczenia 0-żadniego, 1-dolnego, 2-górnego, 3-obu
	iOperPanelButtonsEnableAo:INT;	// Włączenie guzików na panelu operatorskim urządzenia 0-enable, 1-disable
	iInactiveTimeAfterP_FAG:INT;	// Czas na decyzję PASS/FAIL
END_STRUCT
END_TYPE

// ProdLineMachines/S12_Hios/DUTs/stHIOS_TestParameters
TYPE stHIOS_TestParameters :
STRUCT
	iScrewsToFastenAn:INT:= 2;		// Liczba śrub do wkręcenia
	iMinPulseAc:INT:= 80;			// Minimalna liczba impulsów PASS
	iMaxPulseAC:INT:= 140;			// Maksymalna liczba impulsów PASS
END_STRUCT
END_TYPE

// ProdLineMachines/S13_FrontFanPress/DUTs/nFrontFanPress_ErrorCodes
{attribute 'qualified_only'}
{attribute 'strict'}
{attribute 'to_string'}
TYPE nFrontFanPress_ErrorCodes :
(
	// Błędy ogólne
	NoError := 0,
	UnKnownAlarm := 53,						// Niezidentyfikowany alarm maszyny
	UnKnownLock := 54,						// Niezidentyfikowana blokada maszyny
	SelectStationIdError := 230,			// Brak pobranego Id stacji
	StatusSaveError := 89,					// Błąd zapisu statusu
	ResetTimeout := 518,					// Timeout resetu maszyny
	ProgramConfigError := 90,				// Błąd w konfiguracji programu
	SafetySystemNotArmed := 614,			// System safety nie uzbrojony
	NoMachineReactionOnStartSig := 140,		// Brak reakcji na sygnał startu (brak wysunięcia siłownika - brak powietrza itp.)

	TwoHandStartContactsError := 130,		// Błąd styków dwustartu
	WorkPosAchieveTimeout := 131,			// Nie osiągnięto pozycji roboczej w zadanym czasie
	OperInteruptedBeforeWorkPos := 132,		// Za wcześnie puszczono dwustart - część nie wprasowana
	WorkPosLost := 138,						// Utracona pozycja robocza (możliwy brak części)
	StabilizingTimeout := 135,				// Nie ustabilizowano części w kowadle w zadanym czasie
	StabilizerReturnTimeout := 137,			// Nie zwolniono stabilizatora części w zadanym czasie
	HomePosAchieveTimeout := 139			// Nie osiągnięto pozycji bazowej prasy w zadanym czasie
	
);
END_TYPE

// ProdLineMachines/S13_FrontFanPress/DUTs/stFrontFanPress_InOuts
TYPE stFrontFanPress_InOuts :
STRUCT
	st2HandStartIO				: st2HandStartBasic_InOuts;	// Sygnały z układu dwu-startu
	bStabilizerHomePos			AT %I*: BOOL;	
	bPressHomePos				AT %I*: BOOL;	
	bPressWorkPos				AT %I*: BOOL;	
	bStabilizerValve_Q			AT %Q*: BOOL;	
	bPressValve_Q				AT %Q*: BOOL;	
END_STRUCT
END_TYPE

// ProdLineMachines/S18_ManometerCalib/DUTs/nManometerCalibration_ErrorCodes
{attribute 'qualified_only'}
{attribute 'strict'}
{attribute 'to_string'}
TYPE nManometerCalibration_ErrorCodes :
(
	// Błędy ogólne
	NoError := 0,
	UnKnownAlarm := 53,						// Niezidentyfikowany alarm maszyny
	UnKnownLock := 54,						// Niezidentyfikowana blokada maszyny
	ResetTimeout := 518,					// Timeout resetu maszyny
	ProgramConfigError := 90,				// Błąd w konfiguracji programu
	SafetySystemNotArmed := 614,			// System safety nie uzbrojony
	NoMachineReactionOnStartSig := 140,		// Brak reakcji na sygnał startu (brak wysunięcia siłownika - brak powietrza itp.)
	OprationTooLong := 168,					// The operation takes too long time
	// Błędy specyficzne dla maszyny	
	TwoHandStartContactsError := 130,		// Błąd styków dwustartu
	WorkPosAchieveTimeout := 131,			// Nie osiągnięto pozycji roboczej w zadanym czasie
	OperInteruptedBeforeWorkPos := 132,		// Za wcześnie puszczono dwustart - część nie wprasowana
	WorkPosLost := 138,						// Utracona pozycja robocza (możliwy brak części)
	HomePosAchieveTimeout := 139,			// Nie osiągnięto pozycji bazowej w zadanym czasie
	PressureOutOfRange := 141,				// Ciśnienie wzorcowania poza zakresem	
	StationResetRequired := 582				// Wymagany reset stanowiska - wyświetl okno w celu potwierdzenia
);
END_TYPE

// ProdLineMachines/S18_ManometerCalib/DUTs/stManometerCalibration_InOuts
TYPE stManometerCalibration_InOuts :
STRUCT
	st2HandStartIO			: st2HandStartBasic_InOuts;	// Sygnały z układu dwu-startu
	bCompressorSensor		AT %I*: BOOL;	
	bTestFrameHomePos		AT %I*: BOOL;	
	bTestFrameWorkPos		AT %I*: BOOL;	
	bNozzlePusherHomePos	AT %I*: BOOL;	
	bNozzlePusherWorkPos	AT %I*: BOOL;	
	bPressureSensorError	AT %I*: BOOL;	 
	iPressure				AT %I*: INT;
	bTestFrameOpenValve_Q	AT %Q*: BOOL;	
	bTestFrameCloseValve_Q	AT %Q*: BOOL;	
	bNozzlePusherValve_Q	AT %Q*: BOOL;
	bTargetAirValve_Q		AT %Q*: BOOL;
END_STRUCT
END_TYPE

// ProdLineMachines/S18_ManometerCalib/DUTs/stManometerCalibration_TestData
TYPE stManometerCalibration_TestData :
STRUCT
	bPressureCheckingEN: BOOL;		// Flaga włączająca sprawdzanie ciśnienia
	rSettingPressure:REAL;			// Wartość ciśniania do kalibracji
	rSettingPressureDeviation:REAL;	// Dopuszczalna odchyłka ciśnienia +/-	
END_STRUCT
END_TYPE

// ProdLineMachines/Sonictech/Fixtures/NoWeldLock/nStFix_NoWeldLock_ErrorCodes
{attribute 'qualified_only'}
{attribute 'strict'}
{attribute 'to_string'}
TYPE nStFix_NoWeldLock_ErrorCodes :
(
	// Błędy ogólne
	NoError := 0,
	UnKnownAlarm := 53,						// Niezidentyfikowany alarm maszyny
	UnKnownLock := 54,						// Niezidentyfikowana blokada maszyny
	SelectStationIdError := 230,			// Brak pobranego Id stacji
	StatusSaveError := 89,					// Błąd zapisu statusu
	ResetTimeout := 518,					// Timeout resetu maszyny
	ProgramConfigError := 90,				// Błąd w konfiguracji programu
	SafetySystemNotArmed := 614,			// System safety nie uzbrojony
	NoMachineReactionOnStartSig := 140,		// Brak reakcji na sygnał startu (brak wysunięcia siłownika - brak powietrza itp.)
	
	SensorWorkError		:= 183,
	PartsNotWelded	 	:= 272
	);
END_TYPE

// ProdLineMachines/Sonictech/Fixtures/S01_IndicatorAssembly/DUTs/nStFix_S01IndicatorAssy_ErrorCodes
{attribute 'qualified_only'}
{attribute 'strict'}
{attribute 'to_string'}
TYPE nStFix_S01IndicatorAssy_ErrorCodes :
(
	// Błędy ogólne
	NoError := 0,
	UnKnownAlarm := 53,						// Niezidentyfikowany alarm maszyny
	UnKnownLock := 54,						// Niezidentyfikowana blokada maszyny
	ProgramConfigError := 90,				// Błąd w konfiguracji programu
	
	SensorNotReady:= 169,
	IndicatorNotDet:= 170,
	VRingNotDet:= 171,
	VRingIndicatorNotDet:= 172,
	CapNotDet:= 173,
	CapIndicatorNotDet:= 174,
	CapVRingNotDet:= 175,
	CapVRingIndicatorNotDet:= 176	
);
END_TYPE

// ProdLineMachines/Sonictech/Fixtures/S01_IndicatorAssembly/DUTs/stStFix_S01IndicatorAssy_InOut
TYPE stStFix_S01IndicatorAssy_InOut :
STRUCT
	stBalluff 							:stBVS_DigInOut;	// Kamera
	bVacuumON_Q					AT %Q* 	:BOOL;		// Zawór podciśnienia
END_STRUCT
END_TYPE

// ProdLineMachines/Sonictech/Fixtures/S01_IndicatorAssembly/DUTs/stStFix_S01IndicatorAssy_Settings
TYPE stStFix_S01IndicatorAssy_Settings EXTENDS stSonicTech_MachSettings :
STRUCT
	bVacumEN: BOOL;
	bIndicatorCheckEN: BOOL;
	bVRingCheckEN: BOOL;
	bCapCheckEN: BOOL;
	iMaxTrigRepeats:INT;
END_STRUCT
END_TYPE

// ProdLineMachines/Sonictech/Fixtures/S06_CarrierWheelLubrification/V1/DUTs/nStFix_S06CarrierAndWheelAssyGrease_ErrorCodes
{attribute 'qualified_only'}
{attribute 'strict'}
{attribute 'to_string'}
TYPE nStFix_S06CarrierAndWheelAssyGrease_ErrorCodes :
(
	// Błędy ogólne
	NoError := 0,
	UnKnownAlarm := 53,						// Niezidentyfikowany alarm maszyny
	UnKnownLock := 54,						// Niezidentyfikowana blokada maszyny
	ProgramConfigError := 90,				// Błąd w konfiguracji programu
	
	StabilizingTimeout := 135,				// Nie ustabilizowano części w kowadle w zadanym czasie
	StabilizerReturnTimeout := 137			// Nie zwolniono stabilizatora części w zadanym czasie
	
);
END_TYPE

// ProdLineMachines/Sonictech/Fixtures/S06_CarrierWheelLubrification/V1/DUTs/stStFix_S06CarrierAndWheelAssyGrease_InOuts
TYPE stStFix_S06CarrierAndWheelAssyGrease_InOuts :
STRUCT
	bRotationStabilizerClosed	AT %I* :BOOL;		// Ramię stabilizatora pozycja robocza
	bNozzleStabilizerClosed		AT %I* :BOOL;		// Dysza smarownicy pozycja robocza
	bRotationStabValve_Q		AT %Q* :BOOL;		// Zawór stabilizatora	
	bNozzleStabValve_Q			AT %Q* :BOOL;		// Zawór wysunięcia dyszy smarownicy
	bGreaseValve_Q				AT %Q* :BOOL;		// Zawór podający smar
END_STRUCT
END_TYPE

// ProdLineMachines/Sonictech/Fixtures/S06_CarrierWheelLubrification/V1/DUTs/stStFix_S06CarrierAndWheelAssyGrease_Settings
TYPE stStFix_S06CarrierAndWheelAssyGrease_Settings EXTENDS stSonicTech_MachSettings :
STRUCT
	rGreaseApplyTime		: REAL;
END_STRUCT
END_TYPE

// ProdLineMachines/Sonictech/Fixtures/S06_CarrierWheelLubrification/V2/DUTs/nStFix_S06CarrierAndWheelAssyGrease_V2_ErrorCodes
{attribute 'qualified_only'}
{attribute 'strict'}
{attribute 'to_string'}
TYPE nStFix_S06CarrierAndWheelAssyGrease_V2_ErrorCodes :
(
	// Błędy ogólne
	NoError := 0,
	UnKnownAlarm := 53,						// Niezidentyfikowany alarm maszyny
	UnKnownLock := 54,						// Niezidentyfikowana blokada maszyny
	ProgramConfigError := 90,				// Błąd w konfiguracji programu
	
	WheelWrongSide:= 232,					//Koło źle umieszczone 
	LackOfWheel:= 233,						//Brak koła
	RotaryFixtureError:= 234				// Błąd kowadła
);
END_TYPE

// ProdLineMachines/Sonictech/Fixtures/S06_CarrierWheelLubrification/V2/DUTs/stStFix_S06CarrierAndWheelAssyGrease_V2_InOuts
TYPE stStFix_S06CarrierAndWheelAssyGrease_V2_InOuts :
STRUCT
	bRotationStabilizerClosed	AT %I* :BOOL;		// Ramię stabilizatora pozycja robocza
	bNozzleStabilizerClosed		AT %I* :BOOL;		// Dysza smarownicy pozycja robocza
	bRotationStabValve_Q		AT %Q* :BOOL;		// Zawór stabilizatora	
	bNozzleStabValve_Q			AT %Q* :BOOL;		// Zawór wysunięcia dyszy smarownicy
	bGreaseValve_Q				AT %Q* :BOOL;		// Zawór podający smar
	bGreaseSprayValve_Q			AT %Q* :BOOL;		// Zawór natrysku smaru
	stBvsInOut						   : stBVS_DigInOut; //Wejścia i wyjśca dla obsługi kamery
END_STRUCT
END_TYPE

// ProdLineMachines/Sonictech/Fixtures/S06_CarrierWheelLubrification/V2/DUTs/stStFix_S06CarrierAndWheelAssyGrease_V2_Settings
TYPE stStFix_S06CarrierAndWheelAssyGrease_V2_Settings EXTENDS stSonicTech_MachSettings :
STRUCT
	bVacumEN				: BOOL;
	bCheckWheelOrientation	: BOOL;
	rGreaseApplyTime		: REAL;
END_STRUCT
END_TYPE

// ProdLineMachines/Sonictech/Fixtures/S07_CarrierAssyWithPiston/V1/DUTs/nStFix_S07CarrierPistonAssy_ErrorCodes
{attribute 'qualified_only'}
{attribute 'strict'}
{attribute 'to_string'}
TYPE nStFix_S07CarrierPistonAssy_ErrorCodes :
(
	// Błędy ogólne
	NoError := 0,
	UnKnownAlarm := 53,						// Niezidentyfikowany alarm maszyny
	UnKnownLock := 54,						// Niezidentyfikowana blokada maszyny
	ProgramConfigError := 90,				// Błąd w konfiguracji programu
	
	StabilizingTimeout := 135,				// Nie ustabilizowano części w kowadle w zadanym czasie
	StabilizerReturnTimeout := 137			// Nie zwolniono stabilizatora części w zadanym czasie
	
);
END_TYPE

// ProdLineMachines/Sonictech/Fixtures/S07_CarrierAssyWithPiston/V1/DUTs/stStFix_S07CarrierPistonAssy_InOuts
TYPE stStFix_S07CarrierPistonAssy_InOuts :
STRUCT
	bRotationStabilizerClosed	AT %I* :BOOL;		// Ramię stabilizatora pozycja robocza
	bCarierStabilizerOpened		AT %I* :BOOL;		// Dysza smarownicy pozycja robocza
	bRotationStabValve_Q		AT %Q* :BOOL;		// Zawór stabilizatora obrotowego
	bCarierStabValve_Q			AT %Q* :BOOL;		// Zawór stabilizatora jednostki nośnej	
	bVacuumON_Q					AT %Q* :BOOL;		// Zawór podciśnienia
	bVacuumScavenge_Q			AT %Q* :BOOL;		// Zawór przedmuchu dyszy
END_STRUCT
END_TYPE

// ProdLineMachines/Sonictech/Fixtures/S07_CarrierAssyWithPiston/V1/DUTs/stStFix_S07CarrierPistonAssy_Settings
TYPE stStFix_S07CarrierPistonAssy_Settings EXTENDS stSonicTech_MachSettings :
STRUCT
	uiScavengeEveryN 				: UINT:= 30;
	rScavenge_Time_S				: REAL:= 0.7;
END_STRUCT
END_TYPE

// ProdLineMachines/Sonictech/Fixtures/S07_CarrierAssyWithPiston/V2/DUTs/nStFix_S07CarrierPistonAssy_V2_ErrorCodes
{attribute 'qualified_only'}
{attribute 'strict'}
{attribute 'to_string'}
TYPE nStFix_S07CarrierPistonAssy_V2_ErrorCodes :
(
	// Błędy ogólne
	NoError := 0,
	UnKnownAlarm := 53,						// Niezidentyfikowany alarm maszyny
	UnKnownLock := 54,						// Niezidentyfikowana blokada maszyny
	ProgramConfigError := 90,				// Błąd w konfiguracji programu
	
	HeatStampHomeError:= 102,					//Pieczątka pozycja schowana nieosiągnięta
	HeatStampWorkError:= 104,					//Pieczątka pozycja wysunięta nieosiągnięta
	RotaryFixtureError:= 234,					//Błąd mocowania rotacyjneg
	CylinderFixtureError:= 235,					//Błąd mocowania komory tłoka
	DamagedStamp:= 236,							//Uszkodzona stempel układ grzewczy
	HeatStampTempStabWait:= 571					//Oczekiwanie na stabilizację temperatury stempla znakującego
);
END_TYPE

// ProdLineMachines/Sonictech/Fixtures/S07_CarrierAssyWithPiston/V2/DUTs/stMachineSettingsHeatStamp
TYPE stMachineSettingsHeatStamp :
STRUCT
	rHeatStamp_Kp			: REAL;
	rHeatStamp_Ki			: REAL;
	rHeatStamp_Kd			: REAL;
	rHeatStampPID_Cycle		: REAL;
	rHeatStampSetTemperature: REAL;
	rHeatStampAllowDeviation: REAL;
	iHeatStampTime			: INT := 200;
	bHeatStampEnable		: BOOL;
END_STRUCT
END_TYPE

// ProdLineMachines/Sonictech/Fixtures/S07_CarrierAssyWithPiston/V2/DUTs/stStFix_S07CarrierPistonAssy_V2_InOuts
TYPE stStFix_S07CarrierPistonAssy_V2_InOuts :
STRUCT
	bRotationStabilizerClosed	AT %I* :BOOL;		// Ramię stabilizatora pozycja robocza
	bCarierStabilizerOpened		AT %I* :BOOL;		// Dysza smarownicy pozycja robocza
	bCarierStabilizerClosed		AT %I* :BOOL;		// Dysza smarownicy pozycja bazowa
	bHeatStampOpened			AT %I* :BOOL;		// Stempel pozycja wsunieta (bazowa)
	bHeatStampClosed			AT %I* :BOOL;		// Stempel pozycja wysunieta (wykonawcza)
	bStampSafetyGateOpened		AT %I* :BOOL;		// Bramka stempla w pozycji otwartej - można znakować

	bAI_StampTemperature_Error	AT %I* :BOOL;		// Odczyt błędu z modułu
	rHeatStampTemperature		AT %I* :INT;		// Temperatura stempla
	bHeatStampPWMSignal			AT %Q* :BOOL;		// Wysterowanie sygnału dla SSR
	bHeatSafetyGateValve_Q		AT %Q* :BOOL;		// Zawór bramki odchronnej stempla
	bHeatStampValve_Q			AT %Q* :BOOL;		// Zawór stempla
	bRotationStabValve_Q		AT %Q* :BOOL;		// Zawór stabilizatora obrotowego
	bCarierStabValve_Q			AT %Q* :BOOL;		// Zawór stabilizatora jednostki nośnej	
	bVacuumON_Q					AT %Q* :BOOL;		// Zawór podciśnienia
	bVacuumScavenge_Q			AT %Q* :BOOL;		// Zawór przedmuchu dyszy
END_STRUCT
END_TYPE

// ProdLineMachines/Sonictech/Fixtures/S07_CarrierAssyWithPiston/V2/DUTs/stStFix_S07CarrierPistonAssy_V2_Settings
TYPE stStFix_S07CarrierPistonAssy_V2_Settings EXTENDS stSonicTech_MachSettings :
STRUCT
	bHeatStampMakingEnable			: BOOL:= TRUE;
	bHeatStampMarkWhenWeldingActive	: BOOL:= FALSE;
	rHeatStampSetTemperature		: REAL:= 280;
	rHeatStampAllowDeviation		: REAL:= 10;
	rHeatStampMarkingTime			: REAL := 0.5;
//	rHeatStamp_Kp					: REAL; 
//	rHeatStamp_Ki					: REAL;
//	rHeatStamp_Kd					: REAL;
	uiScavengeEveryN 				: UINT:= 30;
	rScavenge_Time_S				: REAL:= 0.7;
END_STRUCT
END_TYPE

// ProdLineMachines/Sonictech/Fixtures/S08_CoolerClosure/V1/nStFix_S08CoolerClosure_ErrorCodes
{attribute 'qualified_only'}
{attribute 'strict'}
{attribute 'to_string'}
TYPE nStFix_S08CoolerClosure_ErrorCodes :
(
	// Błędy ogólne
	NoError := 0,
	UnKnownAlarm := 53,						// Niezidentyfikowany alarm maszyny
	UnKnownLock := 54,						// Niezidentyfikowana blokada maszyny
	ProgramConfigError := 90,				// Błąd w konfiguracji programu
	
	PartStabilizationTimeout := 135,
	PartStabReleaseTimeout := 137
);
END_TYPE

// ProdLineMachines/Sonictech/Fixtures/S08_CoolerClosure/V1/stStFix_S08CoolerClosure_InOuts
TYPE stStFix_S08CoolerClosure_InOuts :
STRUCT
	bRotationStabilizerClosed	AT %I* :BOOL;		// Ramię stabilizatora pozycja robocza
	bRotationStabValve_Q		AT %Q* :BOOL;		// Zawór stabilizatora obrotowego
END_STRUCT
END_TYPE

// ProdLineMachines/Sonictech/Fixtures/S08_CoolerClosure/V2/DUTs/nStFix_S08CoolerClosure_V2_ErrorCodes
{attribute 'qualified_only'}
{attribute 'strict'}
{attribute 'to_string'}
TYPE nStFix_S08CoolerClosure_V2_ErrorCodes :
(
	// Błędy ogólne
	NoError := 0,
	UnKnownAlarm := 53,						// Niezidentyfikowany alarm maszyny
	UnKnownLock := 54,						// Niezidentyfikowana blokada maszyny
	ProgramConfigError := 90,				// Błąd w konfiguracji programu
	
	HeatStampNotDetected:= 240,				//Nie wykryto pieczątki
	BiggerActuatorError:= 241,				//Większy siłownik błąd
	SmallerActuatorError:= 242,				//Mniejszy siłownik błąd
	CoolerActuatorError:= 243,				//Siłownik chłodnicy błąd	
	VisionSensorError := 511			
);
END_TYPE

// ProdLineMachines/Sonictech/Fixtures/S08_CoolerClosure/V2/DUTs/stStFix_S08CoolerClosure_V2_InOuts
TYPE stStFix_S08CoolerClosure_V2_InOuts :
STRUCT
	bBiggerStabilizerOpened		AT %I* :BOOL;		// Większe ramię z elementem pozycja zamknięta
	bBiggerStabilizerClosed		AT %I* :BOOL;		// Większe ramię z elementem pozycja zamknięta
	bSmallerStabilizerOpened	AT %I* :BOOL;		// Mniejsze ramię z elementem pozycja zamknięta
	bSmallerStabilizerClosed	AT %I* :BOOL;		// Mniejsze ramię z elementem pozycja zamknięta
	bCarierUpPosition			AT %I* :BOOL;		// Mocowanie z carrierem pozycja górna
	
	bBiggerStabilizerClose		AT %Q* :BOOL;		// Większe ramię z elementem pozycja zamknięta
	bSmallerStabilizerClose		AT %Q* :BOOL;		// Mniejsze ramię z elementem pozycja zamknięta
	bCarierClose				AT %Q* :BOOL;		// Mocowanie z carrierem pozycja górna
	
	stBvsInOut						   : stBVS_DigInOut; //Wejścia i wyjśca dla obsługi kamery
END_STRUCT
END_TYPE

// ProdLineMachines/Sonictech/Fixtures/S08_CoolerClosure/V2/DUTs/stStFix_S08CoolerClosure_V2_Settings
TYPE stStFix_S08CoolerClosure_V2_Settings EXTENDS stSonicTech_MachSettings :
STRUCT
	bCheckVisionSign		: BOOL:= TRUE;	
	bBiggerActuatorFirst	: BOOL:= FALSE;	
END_STRUCT
END_TYPE

// ProdLineMachines/Sonictech/Fixtures/S10_CoolerCarrierOrifice/stStFix_S10CoolerCarrierOrifice_InOuts
TYPE stStFix_S10CoolerCarrierOrifice_InOuts :
STRUCT
	bRotationStabilizerClosed	AT %I* :BOOL;		// Ramię stabilizatora pozycja robocza
	bStabilizerLockClosed		AT %I* :BOOL;		// Dysza smarownicy pozycja robocza
	bRotationStabValve_Q		AT %Q* :BOOL;		// Zawór stabilizatora obrotowego
	bStabLockValve_Q			AT %Q* :BOOL;		// Zawór stabilizatora jednostki nośnej	
END_STRUCT
END_TYPE

// ProdLineMachines/Sonictech/Fixtures/S16_FixAndFrontFanDetection/DUTs/nStFix_S16PinWeldFfDetection_ErrorCodes
{attribute 'qualified_only'}
{attribute 'strict'}
{attribute 'to_string'}
TYPE nStFix_S16PinWeldFfDetection_ErrorCodes :
(
	// Błędy ogólne
	NoError := 0,
	UnKnownAlarm := 53,						// Niezidentyfikowany alarm maszyny
	UnKnownLock := 54,						// Niezidentyfikowana blokada maszyny
	ResetTimeout := 518,					// Timeout resetu maszyny
	ProgramConfigError := 90,				// Błąd w konfiguracji programu
	NoMachineReactionOnStartSig := 140,		// Brak reakcji na sygnał startu (brak wysunięcia siłownika - brak powietrza itp.)
	
	SensorNotReady:= 169,
	SearchAreaNotVisible:= 180,
	FrontFanNotDetected:= 181,
	SensorWorkError		:= 183,
	PartNotDetectedInFixture:= 190,
	PartsNotWelded	 	:= 272
	);
END_TYPE

// ProdLineMachines/Sonictech/Fixtures/S16_FixAndFrontFanDetection/DUTs/stStFix_S16PinWeldFfDetection_InOuts
TYPE stStFix_S16PinWeldFfDetection_InOuts :
STRUCT
	stBalluff 							:stBVS_DigInOut;	// Kamera
	bEnclosureSensor			AT %I* 	:BOOL;				// Czujnik obudowy
	bRotationStabilizerClosed	AT %I* 	:BOOL;				// Ramię stabilizatora pozycja robocza
	bRotationStabValve_Q		AT %Q* 	:BOOL;				// Zawór stabilizatora obrotowego
	bEnclosureLock_Q			AT %Q* 	:BOOL;				// Blokada obudowy w kowadle
END_STRUCT
END_TYPE

// ProdLineMachines/Sonictech/Fixtures/S16_FixAndFrontFanDetection/DUTs/stStFix_S16PinWeldFfDetection_Settings
TYPE stStFix_S16PinWeldFfDetection_Settings EXTENDS stSonicTech_MachSettings :
STRUCT
	NoWeldLockCheck					: BOOL;
	bIsSearchAreaVisibleCheckEN		: BOOL;
	bFrontFanCheckEN				: BOOL;
END_STRUCT
END_TYPE

// ProdLineMachines/Sonictech/Fixtures/S17_EnclosurePressFix/DUTs/nStFix_S17EnclosureWelding_ErrorCodes
{attribute 'qualified_only'}
{attribute 'strict'}
{attribute 'to_string'}
TYPE nStFix_S17EnclosureWelding_ErrorCodes :
(
	// Błędy ogólne
	NoError := 0,
	ResetTimeout := 518,					// Timeout resetu maszyny
	ProgramConfigError := 90,				// Błąd w konfiguracji programu
	NoMachineReactionOnStartSig := 140,		// Brak reakcji na sygnał startu (brak wysunięcia siłownika - brak powietrza itp.)
	
	PartsNotWelded	 	:= 272,
	HomePositionMissing := 3,
	BasePositionTimeout := 139,
	SensorWorkError		:= 183,
	PartNotDetectedInFixture:= 190,
	TargetPositionTimeout	:= 831
	);
END_TYPE

// ProdLineMachines/Sonictech/Fixtures/S17_EnclosurePressFix/DUTs/stStFix_S17EnclosureWelding_InOuts
TYPE stStFix_S17EnclosureWelding_InOuts :
STRUCT
	bEnclosureSensor 	AT %I*	: 		BOOL;
	bLeftActuatorHome	AT %I*	:		BOOL;
	bRightActuatorHome	AT %I*	:		BOOL;
	bAnvilBottom		AT %I*	:		BOOL;
	bAnvilValve			AT %Q*	:		BOOL;
END_STRUCT
END_TYPE

// ProdLineMachines/Sonictech/SerialCom/DUTs/DataStruct/stSonicTech_SerialStructGenParamsRange
TYPE stSonicTech_SerialStructGenParamsRange :
STRUCT
	byGeneratorType:BYTE:=0;			//
	uiMinGenFrequency:UINT:=0;			//
	uiMaxGenFrequency:UINT:=0;			//
	uiMaxGenPower:UINT:=0;			//
	uiEncoderLength:UINT:=0;			//
END_STRUCT
END_TYPE

// ProdLineMachines/Sonictech/SerialCom/DUTs/DataStruct/stSonicTech_SerialStructProgParams
TYPE stSonicTech_SerialStructProgParams :
STRUCT
	byProgNum:BYTE;					// Numer programu
	byWeldType:BYTE;				// Tryb wykonania zgrzewu - 0 ÷ 4, 0- Czas, 1- Energia, 2- Moc maks., 3- Droga DRM, 4- Droga ABS
	byGenAmplitude:BYTE;			// Amplituda generatora [%] 50 .. 100
	byEmpty:BYTE;
	iMinWeldTime:INT;				// Minimalny czas zgrzewu [ms]
	iMaxWeldTime:INT;				// Maksymalny czas zgrzewu [ms]
	iMinWeldEnergy:INT;				// Minimalna energia zgrzewu [J]
	iMaxWeldEnergy:INT;				// Maksymalna energia zgrzewu [J]
	iMinGenPower:INT;				// Minimalna moc podczas zgrzewu [W]
	iMaxGenPower:INT;				// Maksymalna moc podczas zgrzewu [W]
	iMinDRM:INT;					// Minimalna droga DRM [mm] 1=0,01mm
	iMaxDRM:INT;					// Maksymalna droga DRM [mm] 1=0,01mm
	iMinABS:INT;					// Minimalna droga ABS [mm] 1=0,01mm
	iMaxABS:INT;					// Maksymalna droga ABS [mm] 1=0,01mm
	iMinTrigerPoint:INT;			// Minimalny punkt wyzwalania [mm] 1=0.01mm
	iMaxTrigerPoint:INT;			// Maksymalny punkt wyzwalania [mm] 1=0.01mm
	uiMinWeldFrequency:UINT;		// Minimalna częstotliwość zgrzewu [Hz]
	uiMaxWeldFrequency:UINT;		// Maksymalna częstotliwość zgrzewu [Hz]
	byTrigeringPressure:BYTE;		// Ciśnienie wyzwalania [bar] 1=0.1bar
	byIWeldPressure:BYTE;			// Pierwsze ciśnienie zgrzewania [bar] 1=0.1bar
	bIIWeldPressure_EN:BOOL;		// Status włączenia II ciśnienia zgrzewania 0-wył., 1-zał.
	byIIWeldPressure:BYTE;			// Drugie ciśnienie zgrzewania [bar] 1=0.1bar
	iSwitchWeldPressPoint:INT;		// Punkt przełącznia ciśnienień zgrzewania
	bHoldPressure_EN:BOOL;			// Status włączenia ciśnienia trzymania 0-wył., 1-zał.
	byHoldPressure:BYTE;			// Ciśnienie trzymania [bar] 1=0.1bar
	iHoldTime:INT;					// Czas trzymania [ms]
	bAfterBurstImp_EN:BOOL;			// Status włączenia impulsu po zgrzewie (after nurst) 0-wył., 1-zał.
	bUSTrigerSource:BOOL;			// Żródło wyzwalania ultradźwięków 0-stab. enkodera, 1- sygnał startu
	iAfterBurstImpDelayTime:INT;	// Czas opóźnienia impulsu po zgrzewie [ms]
	iAfterBurstImpTime:INT;			// Czas trwania impulsu po zgrzewie [ms]
	iTrigerDelayTime:INT;			// Czas opóźnienia wyzwolenia [ms]
	bSkanAfterProgChange_EN:BOOL;	// Flaga do uruchomiania po zmianie programu 0- skan. pomijane, 1- skan. uruchamiane
	bEmptyParam_1:BOOL;	
END_STRUCT
END_TYPE

// ProdLineMachines/Sonictech/SerialCom/DUTs/DataStruct/stSonicTech_SerialStructSoftVer
TYPE stSonicTech_SerialStructSoftVer :
STRUCT
	byDriverModel:BYTE:=0;			//1- Thorn+
	byMajorVersion:BYTE:=0;			//
	byMinorVersion:BYTE:=0;			//
	iBuildNumber:INT:=0;			//
END_STRUCT
END_TYPE

// ProdLineMachines/Sonictech/SerialCom/DUTs/DataStruct/stSonicTech_SerialStructWeldParams
TYPE stSonicTech_SerialStructWeldParams :
STRUCT
	byWeldStatus:BYTE;
	byProgramNumber:BYTE;			// Numer wykonanego programu
	byWeldProgType:BYTE;				// Tryb wykonania zgrzewu - 0 ÷ 4
	iWeldTime_ms:INT;			// Minimalny czas zgrzewu [ms]
	iWeldEnergy_J:INT;
	iGenPower_W:INT;
	iDRM_mm:INT;
	iABS_mm:INT;
	iDAHT_mm:INT;
END_STRUCT
END_TYPE

// ProdLineMachines/Sonictech/SerialCom/DUTs/nSonicTech_SerialCmdClasses
{attribute 'qualified_only'}
{attribute 'strict'}
TYPE nSonicTech_SerialCmdClasses :
(
	NoCMD 					:= 0,
	ReadSerialNb			:= 1,	// Funkcja  0x00, Query-SD1, Reply SD2, brak danych wej
	ReadMaxParamsValues 	:= 2,	// Funkcja  0x01, Query-SD1, Reply SD3, brak danych wej
//	PressSetingSonDown	 	:= 3,	// Funkcja  0x02, Query-SD3, Reply SC, Dane wjeściowe to wejście w Menu(1B), wartość ciśnienia(1B)
//	SonotrodePosRead	 	:= 4,	// Funkcja  0x02, Query-SD1, Reply SD3, brak danych wej
	ReadSoftVer 			:= 5,	// Funkcja  0x03, Query-SD1, Reply SD3, brak danych wej
	SetProgNb 				:= 6,	// Funkcja  0x10, Query-SD3, Reply SC, Dane wjeściowe to numer programu(1B)
	ReadProgNb 				:= 7,	// Funkcja  0x10, Query-SD1, Reply SD3, brak danych wej
	SetProgParams 			:= 8,	// Funkcja  0x11, Query-SD2, Reply SC, 
	ReadProgParams 			:= 9,	// Funkcja  0x11
	SetProgName 			:= 10,	// Funkcja  0x12, Query-SD2, Reply SC, Dane wjeściowe to numer programu(1B) i nazwa programu
	ReadProgName 			:= 11,	// Funkcja  0x12, Query-SD3, Reply SD2, Dane wjeściowe to numer programu(1B)
	SetProgParamsEEPROM		:= 12,	// Funkcja  0x13, Query-SD2, Reply SC
	ReadProgParamsEEPROM	:= 13,	// Funkcja  0x13, Query-SD3, Reply SD2, Dane wjeściowe to numer programu(1B)
	ReadWeldParams 			:= 14,	// Funkcja  0x20, Query-SD1, Reply SD2, brak danych wej
	ReadErrorCode 			:= 15	// Funkcja  0x21, Query-SD1, Reply SD3, brak danych wej
);
END_TYPE

// ProdLineMachines/Sonictech/SerialCom/DUTs/nSonicTech_SerialCmdStatus
{attribute 'qualified_only'}
{attribute 'strict'}
TYPE nSonicTech_SerialCmdStatus :
(
	NoStatus := 0,
	Queued := 1,		// Zakolejkowana
	Sended := 2, 		// WYsłana
	WaitForRepply := 3, // Oczekiwanie na odpowiedź potwierdzenie
	CmdSucceed := 4,	// Zakończono OK - odebrano odpowiedź
	CmdError := 5		// Zakońcozno z błędem - brak odpowiedzi itp.
);
END_TYPE

// ProdLineMachines/Sonictech/SerialCom/DUTs/nSonicTech_SerialCmdType
{attribute 'qualified_only'}
{attribute 'strict'}
TYPE nSonicTech_SerialCmdType :
(
	SD1 := 0,
	SD2 := 1,
	SD3 := 2,
	SC := 3
);
END_TYPE

// ProdLineMachines/Sonictech/SerialCom/DUTs/stSonicTech_SerialCMD
// Struktura do komunikacji
TYPE stSonicTech_SerialCMD :
STRUCT
	tTimeStamp				: TIME;								// Znacznik czasowy do sprawdzania timeoutu
	nCmdStatus				: nSonicTech_SerialCmdStatus;	// Dodatkowy debug
	nCmdType				: nSonicTech_SerialCmdClasses;	// Ustalony rodzaj komendy
	pExchangeData 			: POINTER TO BYTE;		// Dane do przekazania do funkcji oraz dane zwrotne po wywołaniu
	uiExchangeDataSize 		: UINT;	// Rozmiar danych
	bySerialAddr			: BYTE;								// Adres szeregowy zgrzewaki do komunikacji
	bSended, bDone, bError: BOOL;
END_STRUCT
END_TYPE
(*
	W momencie dodania rozkazu do kolejki w danych pExchangeData powinny być dane rozakzu. Gdy blok komunikacji
wyślę komendę do zgrzewaki i ustawi flagę bSend do tej zmiennej (pExchangeData) zostaną zapisane dane odczytane ze zgrzewarki 

*)

// ProdLineMachines/Sonictech/Welding Machine/DUTs/nSonicTech_ErrorList
{attribute 'qualified_only'}
//{attribute 'strict'}
{attribute 'to_string'}
TYPE nSonicTech_ErrorList :
(
	// Błędy ogólne
	NoError := 0,
	UnKnownAlarm := 53,						// Niezidentyfikowany alarm maszyny
	UnKnownLock := 54,						// Niezidentyfikowana blokada maszyny
	ResetTimeout := 518,					// Timeout resetu maszyny
	ProgramConfigError := 90,				// Błąd w konfiguracji programu
	SafetySystemNotArmed := 614,			// System safety nie uzbrojony
	NoMachineReactionOnStartSig := 140,		// Brak reakcji na sygnał startu (brak wysunięcia siłownika - brak powietrza itp.)


	
	MemoryError 		:= 1,
	RTC_error 			:= 2,
	HomePositionError 	:= 3,
	TriggerPointError 	:= 4,
	PressureError 		:= 5,
	FrequencyError 		:= 6,
	TimeErrorMin 		:= 7,
	TimeErrorMax 		:= 8,
	EnergyErrorMin 		:= 9,
	EnergyErrorMax 		:= 10,
	PowerErrorMin 		:= 11,
	PowerErrorMax 		:= 12,
	DRM_errorMin 		:= 13,
	DRM_errorMax 		:= 14,
	ABS_errorMin  		:= 15,
	ABS_errorMax  		:= 16,
	MonitTimeExpired 	:= 17,
	NoUltrasound 		:= 18,
	WP_AUX1_Error 		:= 19,
	WP_AUX2_Error 		:= 20,
	HP_AUX1_Error 		:= 21,
	HP_AUX2_Error 		:= 22,
	EmergencyStop 		:= 23,
	ResetIsPressed 		:= 24,
	MemCodingError 		:= 25,
	CondAUX1_Error 		:= 26,
	CondAUX2_Error 		:= 27,
	RewinderError 		:= 28,
	GenCommError 		:= 29,
	ExceedTemperature 	:= 30,
	ExceedProtection 	:= 31,
	GeneratorError 		:= 32,
	ActiveCurtain 		:= 33,
	StartSgnError 		:= 34,
	PowerSupplyError 	:= 35,
	EncoderError 		:= 36,
	ProgramError 		:= 37,
	ParametersError 	:= 38,
	MeasurementError 	:= 39,
	ProgSelError 		:= 40,
	WrongSocket 		:= 41,
	GenModeError 		:= 42,
	GenEnergyError 		:= 43,
	GenPowerError 		:= 44,
	GenParamError 		:= 45,
	NoTransducer 		:= 46,
	GenMultiResonance 	:= 47,
	GenDuringScan  		:= 48,
	ProgGenError 		:= 49,
	SkanGenError 		:= 50,
	Communication_error := 51,
	UndefinedError		:= 52,
	FixtureNoResponse	:= 55,
	FixtureError		:= 57,
	BreakStartSignal 	:= 127,
	SendFrameError		:= 128,
	AUX1OutNotSetUp		:= 129,
	StartSignalToShort 	:= 191,
		
	OutputErrorWeldOk 	:= 86,
	OutputErrorReady 	:= 87,
	OutputErrorError 	:= 88,
	ExtCondNotMet		:= 92
);
END_TYPE

// ProdLineMachines/Sonictech/Welding Machine/DUTs/stSonicTech_DigInOuts
TYPE stSonicTech_DigInOuts :
STRUCT
// Inputs
	bWeld_OK		AT %I*	:BOOL;	// Wygnał o prawidłowym zgrzewie
	bReadyToWelding	AT %I*	:BOOL;	// Sygnał o gotowości do wykonania kolejnego zgrzewu
	bWeldingActive	AT %I*	:BOOL;	// Aktywna generacja ultradźwięków
	bErrorActive	AT %I*	:BOOL;	// Aktywny błąd zgrzewarki ultradźwiękowej
	bStartInput		AT %I*	:BOOL;	// Sygnał z wyjścia na dodatkowy siłownik - nowy zgrzew
// Outputs
	bWorkPermit		AT %Q*	:BOOL;	// Zezwolenie systemu na pracę zgrzewarki ultradźwiękoiwej
	bResetError		AT %Q*	:BOOL;	// Resetowanie błędu zgrzewarki ultradźwiękowej
END_STRUCT
END_TYPE

// ProdLineMachines/Sonictech/Welding Machine/DUTs/stSonicTech_MachSettings
TYPE stSonicTech_MachSettings :
STRUCT
	bSerialCommunicationEN:BOOL:= TRUE;		// Flaga włączająca komunikację szeregową
	bySerialAdress:BYTE:=16#33;				// Adres zgrzewarki ultradźwiękowej domyślnie 51 (0x33)
	bLockWhenOperationsBreaked: BOOL;		// When operation was breaked before achieve safe possition - lock machine
	{attribute 'hide'} 
	bTmp1:BOOL;
END_STRUCT
END_TYPE

// SQL/DUTs/DataSelectDUTs/stSQL_RetDataProdLineStat
TYPE stSQL_RetDataProdLineStat:
STRUCT
	IdLinii : DINT;
	IdStacji : DINT;
	AutoSaveErrors : BOOL;
	IsEOL : BOOL;
	IdOutComposedPart: LINT;
//	AutoControlMachineParams : BOOL;
	CrcSumOfParams:WORD;
	PartCodeNumber:STRING(250);
END_STRUCT
END_TYPE

// SQL/DUTs/DataSelectDUTs/stSQL_RetDataProdMachParams
TYPE stSQL_RetDataProdMachParams:
STRUCT
	StructRawData : ARRAY [1..1000] OF BYTE;
	CRC16sum : INT;
	DataSize: INT;
END_STRUCT
END_TYPE

// SQL/DUTs/DataSelectDUTs/stSQL_RetDataUserRole
TYPE stSQL_RetDataUserRole:
STRUCT
	Role : STRING(500);
	FirstName : STRING(50);
	LastName : STRING(50);
END_STRUCT
END_TYPE

// SQL/DUTs/HMI_DUTs/stSQL_HMI_CoreNodesData
TYPE stSQL_HMI_CoreNodesData :
STRUCT
	iNumber:INT;
	bBusy:BOOL;
	bHangUp:BOOL;
	sLastOperResult:STRING;
END_STRUCT
END_TYPE

// SQL/DUTs/HMI_DUTs/stSQL_HMI_QueueData
TYPE stSQL_HMI_QueueData :
STRUCT
	iNumber:INT;
	sStationName:STRING(5);
	nCmdType:nSQL_CmdTypes;
	bWaitForDataReturn:BOOL;
END_STRUCT
END_TYPE

// SQL/DUTs/nSQL_CmdExecState
{attribute 'qualified_only'}
{attribute 'strict'}
// Funkcjonalnie typ nie potrzebny ale potencjalnie może przydać się przy debugowaniu
TYPE nSQL_CmdExecState :
(
	New:= 0,			// Nowa komenda
	Queued:= 1,			// Komenda została dodana do kolejki
//	Poped:= 2,			// Komenda została pobrana z kolejki - czeka na przetorzenie przez blok - do debugowania
	Processing:= 3,		// Komenda jest przetwarzana przez jądro SQL
	ReSend:= 4,			// Ponowa próba wykonania po błędzie wykonania
	UnQueued:= 5,		// Komenda została usunięta z kolejki gdyż była inna o wyższym priorytecie
	Succeed := 6,		// Komenda wykonana poprawnie, dane pobrane, wyjścia zaktualizowane
	Error:= 7			// Błąd przetwarzania komendy przez serwer SQL
);
END_TYPE

// SQL/DUTs/nSQL_CmdTypes
{attribute 'qualified_only'}
{attribute 'strict'}
{attribute 'to_string'}
// Rodzaje komunikatów które są wysyłane do DB, im wyższy indeks tym większy priorytet.
// Wszystkie metody są zaimplementowane w  bloku - wywoływane są w FB stacji, maszyny lub na zewnątrz
TYPE nSQL_CmdTypes :
(
		// Wyższy numer ma wyższy priorytet wykonania
	None := 0,							// Domyślny - brak akcji
	InsEnergyCons := 1,					// PLC -> 	MySQL DB - Zapisanie w DB aktualnej wartości licznika zużycia energii elektrycznej 
	InsCompressedAirCons := 2,			// PLC -> 	MySQL DB - Zapisanie w DB aktualnej wartości licznika zużycia sprężonego powietrza 
	InsAdditionalError := 3,			// PLC -> 	SQL DB 	- Zapisanie w DB kodu błędu 
	InsExtendedData := 4,				// PLC -> 	MySQL DB - Zapisanie w DB rozszerzonych danych testu/operacji
	InsDefectRelation := 5,				// PLC -> 	SQL DB 	- Zapisanie w DB relacji statusu z kodem alarmu 
	SelLastOperationStatus := 6,		// PLC <- 	SQL DB - Pobranie z DB statusu ostatniej operacji
	SelInsStatusOfOperation := 7,		// PLC <-> 	SQL DB - Zapisanie w DB statusu operacji, pobranie jego identyfikatora 
	SelInsStatusAndExtendedData := 8,	// nieużywane - po podzieleniu zapisu danych na status - dane rozszerzone do innych DB. PLC <-> DB - Zapisanie w DB statusu operacji, danych rozszerzonych, pobranie ID statusu 
	SelMachineParamsCRC := 9,			// PLC <- 	SQL DB  - Pobranie aktualnej sumy CRC dla zestawu stacja + komponent
	SelMachineParams := 10,				// PLC <- 	SQL DB- Pobranie aktualnych parametrów pracy maszyny 
	InsMachineParams := 11,				// PLC -> 	SQL DB - Zapisanie w DB aktualnych parametrów pracy maszyny 
	SelUserRole := 12,					// PLC <- 	SQL DB- Zapytanie o stanowisko/poziom dostępu na podst. numeru ID
	SelStationId := 13					// PLC <- 	SQL DB- Pobranie ID stanowiska, czy AutoSaveError itp.
);
END_TYPE

// SQL/DUTs/nSQL_ErrorCodes
{attribute 'qualified_only'}
{attribute 'strict'}
TYPE nSQL_ErrorCodes :
(
	// Common errors	
	NoError := 0,										// Brak błędu
	UnKnownAlarm := 53,									// Niezidentyfikowany alarm maszyny
	UnKnownLock := 54,									// Niezidentyfikowana blokada maszyny
	ProgramError := 90,									// Błąd w konfiguracji oprogramowania - zerowy wskaźńik itp
	AddBadPointer := 1,									// Dodanie nowego zapytania SQL - zerowy wskaźnik, zapytanie pominięte
	AddNewOperatorFail := 2,							// Błąd alokacji pamięci dynamicznej - brak miejsca w pamięci itp.
	AddNewNoSpaceForAddPriority := 3,					// Kolejka zapytań pełna, brak miejsca dla zapytania o danym priorytecie
	AddNewFailedMasterErrorAtCore := 4,					// Poważny błąd związany z DB - brak licencji itp. - dalsza komunikacja nie ma sensu do czasu reakcji na błąd
	
	SQL_SelectParamsError:= 106,
	SQL_InsertParamsError:= 107
);
END_TYPE

// SQL/DUTs/nSQL_UserRoles
{attribute 'qualified_only'}
//{attribute 'strict'}
{attribute 'to_string'}
TYPE nSQL_UserRoles :
(
	NONE:= 0,
	Unspecified:= 1,
	Operator := 2,
	Quality := 3,
	RDChem := 4,
	Trainer := 5,
	Maintenance := 6,
	LineLeader := 7,
	ShiftLeader := 8,
	Supervisor := 9,
	RD := 10,
	Engineering := 11,
	AdminUser:= 12
);
END_TYPE

// SQL/DUTs/stSQL_ClientNode
{attribute 'enable_dynamic_creation'}
TYPE stSQL_ClientNode :
STRUCT
	nCmdType:nSQL_CmdTypes;				// Typ komendy - od niego zależy priorytet wysłania
	nCmdState:nSQL_CmdExecState;		// Stanus przetwarzania komendy - tylko do celów informacyjnych
	sStation: STRING(15);				// Numer linii i stanowiska
	udiReadStartIndex: UDINT;			// Future reference - Indeks pierwszego rekordu do odczytu (zwykle 0)
	udiRecordCount: UDINT;				// Future reference - info ile linijek odczytać
	bWaitForDataReturn:BOOL;			// Jeśli TRUE - blok klienta czeka na wykonanie rozkazu (operowanie na strukturach klienta), FALSE- klient dodaje komende do kolejki oraz idzie dalej bez blokowania (tworzona jest dynamicznie kopia zapytania)
	byExecutingNodeNb:BYTE;				// Numer węzła przetwarzającego komendę - debugging
	sCmdExpression:STRING(1023);		// komenda SQL do wykonania
	stStatusSaveParams: stSQL_SaveStatustParams;		// 
	pReturnedData:POINTER TO BYTE;		// Jeśli komenda zwraca dane przypisz wskaźnik do danych zwrotnych (zmienna bWaitForDataReturn musi być ustawiona)
	uiReturnedDataSize:UINT;			// Rozmiar struktury danych zwrotnych
	bSQL_LifeBit, bSQL_Busy, bSQL_Done, bSQL_OK: BOOL := FALSE;	// Stany przetwarzania komendy + lifebit (Core ustawia lifebit podczas przetwarzania)
	udiLEventId: UDINT;
	rCmdExecTimeMS: REAL;
	sEventText:STRING;
END_STRUCT
END_TYPE

// SQL/DUTs/stSQL_SaveStatustParams
TYPE stSQL_SaveStatustParams :
STRUCT
	didLineStation	: DINT;		// From database
	byStatus		: BYTE;		// 0 or 1
	iMachineNb		: INT;		// Machine number
	byIsHidden		: BYTE;		// IsHidden flag for status
	byIsTestMode	: BYTE;		// IsTestMode
	lrQuantity		: LREAL;	// Guantity of items
END_STRUCT
END_TYPE

// VisionSensors/Balluff BVS/stBVS_DigInOut
TYPE stBVS_DigInOut :
STRUCT
	bDI_TriggerSignal AT %I*:BOOL;		// Detekcja zakończona - wyjścia aktualne (zmiana stanu) (Wyjście nr 4 ustawione jako Toogle)
	bDI_Input_1 AT %I*:BOOL;			// Wejście 1 (Baluff wyjście 1) - przypisane zgodnie z detekcją
	bDI_Input_2 AT %I*:BOOL;			// Wejście 2 (Baluff wyjście 2) - przypisane zgodnie z detekcją
	bDI_Input_3 AT %I*:BOOL;			// Wejście 3 (Baluff wyjście 3) - przypisane zgodnie z detekcją
	bDO_InputSelect AT %Q*:BOOL;		// Przełączanie programu w czujniku
	bDO_Trigger AT %Q*:BOOL;			// Ręczne wyzwolenie detekcji w czujniku
END_STRUCT
END_TYPE

// VisionSensors/Cognex/stCognexIS280_DigInOut
// Cognex nie synchronizuje wyjść detekcji oraz wyjścia busy więc trzeba ustawić czas trwania pulsu na min. 200ms
TYPE stCognexIS280_DigInOut :
STRUCT
	bIn0 AT %I*:BOOL;				// Sygnał w In-Sight Out0 - zwykle używane jako sygnał Busy
	bIn1 AT %I*:BOOL;				// Sygnał w In-Sight Out1 - Wejście detekcji 1
	bInOut2 AT %I*:BOOL;			// Sygnał w In-Sight Out2 - Wejście detekcji 2
	bInOut3 AT %I*:BOOL;			// Sygnał w In-Sight Out3 - Wejście detekcji 3
	bOut0_Trigger AT %Q*:BOOL;		// Sygnał w In-Sight In0 - Wyjście wyzowlenia detekcji
	bOut1 AT %Q*:BOOL;				// Sygnał w In-Sight In1 - Wyjście zwykle nie używane
END_STRUCT
END_TYPE

// VisionSensors/Keyence/IV3/stKeyenceIV3_DigInOut
TYPE stKeyenceIV3_DigInOut :
STRUCT
	bDI_OUT1 AT %I*:BOOL;			// Sygnał Busy - wyjścia aktualne (zmiana stanu)
	bDI_OUT2 AT %I*:BOOL;				// Wyjście 2 - przypisane zgodnie z detekcją
	bDI_OUT3 AT %I*:BOOL;				// Wyjście 3 - przypisane zgodnie z detekcją
	bDI_OUT4 AT %I*:BOOL;				// Wyjście 4- przypisane zgodnie z detekcją
	bDI_OUT5 AT %I*:BOOL;				// Wyjście 5- przypisane zgodnie z detekcją
	bDI_OUT6 AT %I*:BOOL;				// Wyjście 6- przypisane zgodnie z detekcją
	bDO_IN1_Trigger AT %Q*:BOOL;		// Zewnętrzne wyzwolenie detekcji w czujniku
	bDO_IN2 AT %Q*:BOOL;				// Wejście swobodnie programowalnw w czujniku
	bDO_IN3 AT %Q*:BOOL;				// Wejście swobodnie programowalnw w czujniku
END_STRUCT
END_TYPE

// VisionSensors/Keyence/stKeyence_DigInOut
TYPE stKeyence_DigInOut :
STRUCT
	bDI_OUT1_Busy AT %I*:BOOL;			// Sygnał Busy - wyjścia aktualne (zmiana stanu)
	bDI_OUT2 AT %I*:BOOL;				// Wyjście 2 - przypisane zgodnie z detekcją
	bDI_OUT3 AT %I*:BOOL;				// Wyjście 3 - przypisane zgodnie z detekcją
	bDI_OUT4 AT %I*:BOOL;				// Wyjście 4- przypisane zgodnie z detekcją
	bDO_IN1_Trigger AT %Q*:BOOL;		// Zewnętrzne wyzwolenie detekcji w czujniku
	bDO_IN2 AT %Q*:BOOL;				// Wejście swobodnie programowalnw w czujniku
	bDO_IN3 AT %Q*:BOOL;				// Wejście swobodnie programowalnw w czujniku
	bDO_IN4 AT %Q*:BOOL;				// Wejście swobodnie programowalnw w czujniku
	bDO_IN5 AT %Q*:BOOL;				// Wejście swobodnie programowalnw w czujniku
	bDO_IN6 AT %Q*:BOOL;				// Wejście swobodnie programowalnw w czujniku
END_STRUCT
END_TYPE

// VisionSensors/stVisionSensor_DigInOut
// Cognex nie synchronizuje wyjść detekcji oraz wyjścia busy więc trzeba ustawić czas trwania pulsu na min. 200ms
TYPE stVisionSensor_DigInOut :
STRUCT
	bIn0 AT %I*:BOOL;				// Sygnał Out0 - zwykle używane jako sygnał Busy
	bIn1 AT %I*:BOOL;				// Sygnał Out1 - Wejście detekcji 1
	bInOut2 AT %I*:BOOL;			// Sygnał Out2 - Wejście detekcji 2
	bInOut3 AT %I*:BOOL;			// Sygnał Out3 - Wejście detekcji 3
	bOut0_Trigger AT %Q*:BOOL;		// Sygnał In0 - Wyjście wyzowlenia detekcji
	bOut1 AT %Q*:BOOL;				// Sygnał In1 - Wyjście zwykle nie używane
	bOut2 AT %Q*:BOOL;				// Sygnał In2 - Wyjście zwykle nie używane
	bOut3 AT %Q*:BOOL;				// Sygnał In3 - Wyjście zwykle nie używane
	bOut4 AT %Q*:BOOL;				// Sygnał In4 - Wyjście zwykle nie używane
END_STRUCT
END_TYPE

// GVL_Aircom
{attribute 'qualified_only'}
VAR_GLOBAL CONSTANT
	sLogsPath:STRING:= 'C:\Logs PLC\';
	// Określenie wyglądu dla każdego rodzaju alarmu - 
	iAlarmClassesQty:INT:= 7;
	astAlarmColorTable:ARRAY [1 .. iAlarmClassesQty] OF stAlarmRowAppearanceData:= [
		(sFontName:='Arial', iFontSize:=10, dwFontFlags:=0, dwTextColor:=16#FF404040, dwAlignmentFlags:=0, dwBackgroundColor:=16#FFCDCDCD, dwFrameColor:=16#FF585858, iFrameWidth:= 1),	// Info
		(sFontName:='Arial', iFontSize:=10, dwFontFlags:=0, dwTextColor:=16#FF404040, dwAlignmentFlags:=0, dwBackgroundColor:=16#FFCDCDCD, dwFrameColor:=16#FF585858, iFrameWidth:= 1),	// Warning
		(sFontName:='Arial', iFontSize:=10, dwFontFlags:=0, dwTextColor:=16#FF404040, dwAlignmentFlags:=0, dwBackgroundColor:=16#FFCDCDCD, dwFrameColor:=16#FF585858, iFrameWidth:= 1),	// Error
		(sFontName:='Arial', iFontSize:=10, dwFontFlags:=0, dwTextColor:=16#FF404040, dwAlignmentFlags:=0, dwBackgroundColor:=16#FFCDCDCD, dwFrameColor:=16#FF585858, iFrameWidth:= 1),	// Quality
		(sFontName:='Arial', iFontSize:=10, dwFontFlags:=0, dwTextColor:=16#FF404040, dwAlignmentFlags:=0, dwBackgroundColor:=16#FFCDCDCD, dwFrameColor:=16#FF585858, iFrameWidth:= 1),	// Maintenance
		(sFontName:='Arial', iFontSize:=10, dwFontFlags:=0, dwTextColor:=16#FF404040, dwAlignmentFlags:=0, dwBackgroundColor:=16#FFCDCDCD, dwFrameColor:=16#FF585858, iFrameWidth:= 1),	// IT
		(sFontName:='Arial', iFontSize:=10, dwFontFlags:=0, dwTextColor:=16#FF404040, dwAlignmentFlags:=0, dwBackgroundColor:=16#FFCDCDCD, dwFrameColor:=16#FF585858, iFrameWidth:= 1)	// Developer
		]; 	
END_VAR

VAR_GLOBAL PERSISTENT
	sCurrentLanguage:STRING(10);
END_VAR

VAR_GLOBAL 
	bInit: BOOL:=TRUE;
	bInitDone: BOOL:=FALSE;
	bWritePersistent: BOOL;						// Save persistent data
	bWritePersistentDelay_1M: BOOL;				// Save persistent data
	stAC_DT_Data: stAircomTimeStruct;			// Time data
	fbRand: DRAND;
	
	bUserLogged: BOOL;
	nUserRole: nSQL_UserRoles;
	sUserName: STRING;
	bPermissionGranted: BOOL;
	fbFormatString: FB_FormatString;
	bSonicTechSerialComDebug: BOOL:= FALSE;		// If TRUE Sonictech seriall com dont return error when communication error.
END_VAR

// Common/2HandStart/BasicVer/fb2HandStartBasic
FUNCTION_BLOCK fb2HandStartBasic
VAR_IN_OUT
	stInOutsData	: st2HandStartBasic_InOuts;
END_VAR
VAR_INPUT
	tDeltaDwuStart	: TIME := T#200MS;
END_VAR
VAR_OUTPUT
	bStartSig		: BOOL;
END_VAR
VAR
	fbStartFilter:fbBinaryFilter;
	fbTON_Dwustart: TON;
END_VAR

tDeltaDwuStart := LIMIT(T#120MS,tDeltaDwuStart,T#800MS);
fbStartFilter(IN:= NOT stInOutsData.bLeftStart_NC AND stInOutsData.bRightStart_NO AND NOT fbTON_Dwustart.Q, tON :=T#30MS, tOFF := T#30MS);
fbTON_Dwustart(IN:= (NOT stInOutsData.bLeftStart_NC OR stInOutsData.bRightStart_NO) AND NOT fbStartFilter.IN, PT := tDeltaDwuStart- T#30MS);
bStartSig := fbStartFilter.Q;

END_FUNCTION_BLOCK

// Common/fbBinaryFilter
FUNCTION_BLOCK fbBinaryFilter
VAR_INPUT
	IN:BOOL;		// Input signal
	tON:TIME;		// Time to set output
	tOFF:TIME;		// Time to reset output
	bReset:BOOL;	// Set output to 0 without any circumstances
END_VAR
VAR_OUTPUT
	Q:BOOL;			// Filtered signal
	RTrig:BOOL;		// Rising edge of Q signal
	FTrig:BOOL;		// Falling edge of Q signal
END_VAR
VAR
	fbTON:TON;
	Q_Mem: BOOL;
END_VAR

IF Q THEN	// Waiting desired time
	fbTON(IN:= NOT fbTON.Q AND NOT bReset AND NOT IN, PT:= tOFF);	
ELSE
	fbTON(IN:= NOT fbTON.Q AND NOT bReset AND IN, PT:= tON);
END_IF
Q := (Q XOR fbTON.Q) AND NOT bReset;	// Switch output
RTrig := Q AND NOT Q_Mem;				// Rtrig calculation
FTrig := NOT Q AND Q_Mem;				// Ftrig calculation
Q_Mem := Q;								// Memorising the Q bit

END_FUNCTION_BLOCK

// Common/2HandStart/fb2HandStart
FUNCTION_BLOCK fb2HandStart
VAR_IN_OUT
	stInOutsData	: st2HandStart_InOuts;
END_VAR
VAR_INPUT
	bNoNcMode		: BOOL:= FALSE;		// Jeśli true bierz pod uwagę styki NC z lewego i NO z prawego przycisku
	b2xNoMode		: BOOL:= FALSE;		// Jeśli true bierz pod uwagę tylko styki NO (brak podłączonych styków NC)
	tDeltaDwuStart	: TIME := T#200MS;
	bReset			: BOOL;
END_VAR
VAR_OUTPUT
	bStartSig		: BOOL;
	bContactsError	: BOOL;
END_VAR
VAR
	fbStartFilter:fbBinaryFilter;
	fbTON_Dwustart: TON;
	fbTON_ContactErrorL, fbTON_ContactErrorP:TON;
	tLastNoNcContactsDiffTimeL, tLastNoNcContactsDiffTimeP:TIME;
	bContactsErrorL, bContactsErrorP: BOOL;
	bResetMem: BOOL;
END_VAR

IF NOT b2xNoMode AND NOT bNoNcMode THEN
	bContactsErrorL := (stInOutsData.bLeftStart_NO AND stInOutsData.bLeftStart_NC) 
						OR ( NOT stInOutsData.bLeftStart_No AND NOT stInOutsData.bLeftStart_NC); 
	bContactsErrorP := (stInOutsData.bRightStart_NO AND stInOutsData.bRightStart_NC ) 
						OR ( NOT stInOutsData.bRightStart_NO AND NOT stInOutsData.bRightStart_NC);
	IF NOT bContactsErrorL AND fbTON_ContactErrorL.IN THEN
		tLastNoNcContactsDiffTimeL := fbTON_ContactErrorL.ET;
	END_IF
	IF NOT bContactsErrorP AND fbTON_ContactErrorP.IN THEN
		tLastNoNcContactsDiffTimeP := fbTON_ContactErrorP.ET;
	END_IF
	fbTON_ContactErrorL(IN:= bContactsErrorL, PT:= tDeltaDwuStart);
	fbTON_ContactErrorP(IN:= bContactsErrorP, PT:= tDeltaDwuStart);
	bContactsError S= fbTON_ContactErrorL.Q OR fbTON_ContactErrorP.Q;
	bContactsError R= bReset AND NOT bResetMem;
	bResetMem := bReset;
	fbStartFilter(IN:= stInOutsData.bLeftStart_NO AND stInOutsData.bRightStart_NO AND NOT fbTON_Dwustart.Q, tON :=T#30MS, tOFF := T#30MS);
	fbTON_Dwustart(IN:= (stInOutsData.bLeftStart_NO OR stInOutsData.bRightStart_NO) AND NOT fbStartFilter.IN, PT := tDeltaDwuStart);
//	bStartSig := stInOutsData.bLeftStart_NO AND stInOutsData.bRightStart_NO AND (NOT fbTON_Dwustart.Q OR bStartSig);
ELSIF bNoNcMode THEN
	bContactsError := FALSE;
//	bStartSig := NOT stInOutsData.bLeftStart_NC AND stInOutsData.bRightStart_NO AND NOT fbTON_Dwustart.Q;
	fbStartFilter(IN:= NOT stInOutsData.bLeftStart_NC AND stInOutsData.bRightStart_NO AND NOT fbTON_Dwustart.Q, tON :=T#30MS, tOFF := T#30MS);
	fbTON_Dwustart(IN:= (NOT stInOutsData.bLeftStart_NC OR stInOutsData.bRightStart_NO) AND NOT fbStartFilter.IN, PT := tDeltaDwuStart+ T#30MS);
ELSIF b2xNoMode THEN
	bContactsError := FALSE;
//	bStartSig := stInOutsData.bLeftStart_NO AND stInOutsData.bRightStart_NO AND NOT fbTON_Dwustart.Q;
	fbStartFilter(IN:= stInOutsData.bLeftStart_NO AND stInOutsData.bRightStart_NO AND NOT fbTON_Dwustart.Q, tON :=T#30MS, tOFF := T#30MS);
	fbTON_Dwustart(IN:= (stInOutsData.bLeftStart_NO OR stInOutsData.bRightStart_NO) AND NOT fbStartFilter.IN, PT := tDeltaDwuStart+ T#30MS);
ELSE
	fbStartFilter(IN:= FALSE, bReset := TRUE);
	bContactsError := FALSE;	 
END_IF
bStartSig := fbStartFilter.Q;

END_FUNCTION_BLOCK

// Common/Actuator/fbActuator
FUNCTION_BLOCK fbActuator
VAR_INPUT
	bI_Control_Ready:BOOL;					// Sygnał gotowości sterowania, sygnały otwórz/zamknij ustawiane tylko gdy jest gotowość
	bI_Opened:BOOL;							// Sygnał z krańcówki otwarcia
	bI_Closed:BOOL;							// Sygnał z krańcówki zamknięcia
	bI_MANUAL_CMD:BOOL;						// Sygnał o ręcznym trybie sterowania
	bI_OpenInterlock:BOOL;					// Sygnał blokady otwierania zaworu/napędu (kolizja z innymi elementami) - powiązane z bI_RespectInterlockInMAN
	bI_CloseInterlock:BOOL;					// Sygnał blokady zamykania zaworu/napędu (kolizja z innymi elementami) - powiązane z bI_RespectInterlockInMAN
	bI_SusteinOpenPos:BOOL;					// Po dojściu do pozycji zadanej podtrzymaj sygnał sterujący - stosować np. dla zaworów 5/2 w celu podtrzymania zamknięcia
	bI_SusteinClosePos:BOOL;				// Po dojściu do pozycji zadanej podtrzymaj sygnał sterujący - stosować np. dla zaworów 5/2 w celu podtrzymania zamknięcia
	bI_RespectInterlockInMAN:BOOL:= TRUE;	// W trybie manualnym uwzględniaj interlocki czy nie
	bI_ResetErr:BOOL;
	bAllowOverCrossPosition:BOOL;			// Ustawiaj sygnał otwórz/zamknij gdy ustawi się odpowiednia krańcówka oraz gdy aktywny sygnał sterujący (zejście z krańcówki przy podtrzymaniu nie powoduje zaniku sygnału otwarcia/zamknięcia)
	bEnPossLossAlarm:BOOL:= FALSE;
	rI_OpenTime:REAL;
	rI_CloseTime:REAL;
	sActuatorId:STRING(30):= 'fbAct';
	sLangId:STRING(2);
	fbAlarmTab:REFERENCE TO fbAlarmSlaveTable;
END_VAR
VAR_OUTPUT
	bQ_Opened:BOOL;
	bQ_Closed:BOOL;
	bDO_Open:BOOL:=FALSE;
	bDO_Close:BOOL:=FALSE;
	bCmdActive:BOOL;
	bInMovement:BOOL;
END_VAR
VAR
	fbTON_OpenTimer:TON;
	fbTON_CloseTimer:TON;
	fbRTrig_Open:R_TRIG;
	fbRTrig_Close:R_TRIG;	
	fbRTrig_Ctr_Open:R_TRIG;
	fbRTrig_Ctr_Close:R_TRIG;	
	fbFTRIG_OpenPosition: F_TRIG;
	fbFTRIG_ClosePosition: F_TRIG;
	bOpen_Cmd: BOOL;
	bClose_Cmd: BOOL;
	fbFTrig_Opened: F_TRIG;
	fbFTrig_Closed: F_TRIG;
	rOpenMeanTime: REAL;
	rCloseMeanTime: REAL;
	bOpenTimeExceedAlSend: BOOL;
	bCloseTimeExceedAlSend: BOOL;
	bSwitchesErrorAlSend: BOOL;
	
	fbTON_controlReady: TON;
END_VAR

VAR PERSISTENT
	diNbOfOperations:DINT;
END_VAR


// Wsuń/zamknij
bClose_Cmd R= ( (bI_Closed OR fbTON_CloseTimer.Q) AND NOT bI_SusteinClosePos) OR NOT bI_Control_Ready;
//bClose_Cmd R= ( (bI_Closed OR (fbTON_CloseTimer.Q AND FALSE)) AND NOT bI_SusteinClosePos) OR NOT bI_Control_Ready;
bDO_Close := bClose_Cmd AND (SEL(bI_MANUAL_CMD, NOT bI_CloseInterlock, NOT (bI_CloseInterlock AND bI_RespectInterlockInMAN)) OR bQ_Closed);
bDO_Open R= bDO_Close;

// Wysuń/otwórz
bOpen_Cmd R= ( (bI_Opened OR fbTON_OpenTimer.Q) AND NOT bI_SusteinOpenPos) OR NOT bI_Control_Ready;
//bOpen_Cmd R= ( (bI_Opened OR (fbTON_OpenTimer.Q AND FALSE)) AND NOT bI_SusteinOpenPos) OR NOT bI_Control_Ready;
bDO_Open := bOpen_Cmd AND (SEL(bI_MANUAL_CMD, NOT bI_OpenInterlock, NOT (bI_OpenInterlock AND bI_RespectInterlockInMAN)) OR bQ_Opened);
bDO_Close R= bDO_Open;

// Określenie sygnałów zamknięcia/otwarcia
fbFTrig_Opened (CLK := bI_Opened);
fbFTrig_Closed (CLK := bI_Closed);
IF bAllowOverCrossPosition THEN
	bQ_Opened R= (NOT bDO_Open AND fbFTrig_Opened.Q) OR bI_Closed; 
	bQ_Closed R= (NOT bDO_Close AND fbFTrig_Closed.Q) OR bI_Opened;
	bQ_Opened S= bI_Opened;
	bQ_Closed S= bI_Closed;
ELSE
	bQ_Opened := bI_Opened;
	bQ_Closed := bI_Closed; 
END_IF
bCmdActive := FALSE;

// Kontrola czasu pracy siłownika
IF fbTON_OpenTimer.IN AND NOT (bDO_Open AND NOT bQ_Opened) AND NOT fbTON_OpenTimer.Q THEN
	fMeanFilter(rInputValue := TIME_TO_REAL(fbTON_OpenTimer.ET), rDelta := 10.0, rMeanValue := rOpenMeanTime);
END_IF
fbTON_OpenTimer(IN := bDO_Open AND NOT bQ_Opened, PT:= REAL_TO_TIME(1000.0*rI_OpenTime));

IF fbTON_CloseTimer.IN AND NOT (bDO_Close AND NOT bQ_Closed) AND NOT fbTON_CloseTimer.Q THEN
	fMeanFilter(rInputValue := TIME_TO_REAL(fbTON_CloseTimer.ET), rDelta := 10.0, rMeanValue := rCloseMeanTime);
END_IF
fbTON_CloseTimer(IN := bDO_Close AND NOT bQ_Closed, PT:= REAL_TO_TIME(1000.0*rI_CloseTime));

bInMovement:= fbTON_OpenTimer.IN OR fbTON_CloseTimer.IN;

// Kontrola błędów w pracy
fbTON_controlReady(IN:= bI_Control_Ready, PT:= T#5S);		// Alarmuj tylko po powrocie sygnału gotowości napędów

// Błąd osiągnięcia pozycji otwórz w odpowiednim czasie
IF fbTON_OpenTimer.Q AND fbTON_controlReady.Q AND __ISVALIDREF(fbAlarmTab) THEN
	IF NOT bOpenTimeExceedAlSend THEN
		fbAlarmTab.mPushRow(nAlarmClass:= enAlarmClasses.Error, sMachineId := sActuatorId, sEventDesc := 'Open time exceeded, open position not achieved', dwErrorId := 0);
		bOpenTimeExceedAlSend := TRUE;
	END_IF
ELSE
	bOpenTimeExceedAlSend := FALSE;
END_IF

// Błąd osiągnięcia pozycji zamknij w odpowiednim czasie
IF fbTON_CloseTimer.Q AND fbTON_controlReady.Q AND __ISVALIDREF(fbAlarmTab) THEN
	IF NOT bCloseTimeExceedAlSend THEN
		fbAlarmTab.mPushRow(nAlarmClass:= enAlarmClasses.Error, sMachineId := sActuatorId, sEventDesc := 'Close time exceeded, close position not achieved', dwErrorId := 0);
		bCloseTimeExceedAlSend := TRUE;
	END_IF
ELSE
	bCloseTimeExceedAlSend := FALSE;
END_IF

// Utracenie pozycji otwarcia
fbFTRIG_OpenPosition(CLK:= bQ_Opened);
IF fbFTRIG_OpenPosition.Q AND NOT bDO_Open AND NOT bDO_Close AND fbTON_controlReady.Q AND bEnPossLossAlarm AND __ISVALIDREF(fbAlarmTab) THEN
	fbAlarmTab.mPushRow(nAlarmClass:= enAlarmClasses.Error, sMachineId := sActuatorId, sEventDesc := 'Loss open position', dwErrorId := 0);
END_IF

// Utracenie pozycji zamknięcia
fbFTRIG_ClosePosition(CLK:= bQ_Closed);
IF fbFTRIG_ClosePosition.Q AND NOT bDO_Open AND NOT bDO_Close AND fbTON_controlReady.Q AND bEnPossLossAlarm AND __ISVALIDREF(fbAlarmTab) THEN
	fbAlarmTab.mPushRow(nAlarmClass:= enAlarmClasses.Error, sMachineId := sActuatorId, sEventDesc := 'Loss close position', dwErrorId := 0);
END_IF

// Kontrola pracy krańcówek
fbRTrig_Open(CLK := bI_Opened);
fbRTrig_Close(CLK := bI_Closed);

IF ((bDO_Open AND fbRTrig_Close.Q AND NOT bAllowOverCrossPosition) OR (bDO_Close AND fbRTrig_Open.Q AND NOT bAllowOverCrossPosition) OR (bI_Opened AND bI_Closed) AND fbTON_controlReady.Q ) AND __ISVALIDREF(fbAlarmTab) THEN
	IF NOT bSwitchesErrorAlSend THEN
		fbAlarmTab.mPushRow(nAlarmClass:= enAlarmClasses.Error, sMachineId := sActuatorId, sEventDesc := 'End stops error', dwErrorId := 0);
	END_IF
ELSE
	bSwitchesErrorAlSend := FALSE;
END_IF

// Ilość cykli pracy
fbRTrig_Ctr_Open (CLK := bDO_Open);
fbRTrig_Ctr_Close (CLK := bDO_Close);
IF fbRTrig_Ctr_Open.Q OR fbRTrig_Ctr_Close.Q THEN
	diNbOfOperations := diNbOfOperations+1;
END_IF

METHOD mClose : BOOL
VAR_INPUT
	bManCtrl:BOOL;
END_VAR
IF bManCtrl THEN
	bClose_Cmd S= bI_MANUAL_CMD;
ELSE
	bClose_Cmd S= NOT bI_MANUAL_CMD;
END_IF
bOpen_Cmd R= bClose_Cmd;
bCmdActive := TRUE;
(*bResult := bClose_Cmd;
IF bManCtrl THEN
	bClose_Cmd S= bI_MANUAL_CMD AND NOT (bI_CloseInterlock AND bI_RespectInterlockInMAN);
ELSE
	bClose_Cmd S= NOT bI_MANUAL_CMD AND NOT bI_CloseInterlock;
END_IF
*)
END_METHOD

METHOD mOpen : BOOL
VAR_INPUT
	bManCtrl:BOOL;
END_VAR
IF bManCtrl THEN
	bOpen_Cmd := bI_MANUAL_CMD;
ELSE
	bOpen_Cmd := NOT bI_MANUAL_CMD;
END_IF
bClose_Cmd R= bOpen_Cmd;
bCmdActive := TRUE;
//bResult := bClose_Cmd;
END_METHOD

METHOD mReset : BOOL
VAR_INPUT
END_VAR
// Reset błędów 
fbTON_OpenTimer(IN:= FALSE);
fbTON_CloseTimer(IN:= FALSE);
END_METHOD

METHOD mStop : BOOL
VAR_INPUT
	bManCtrl:BOOL;
END_VAR
IF bManCtrl THEN
	bOpen_Cmd R= bDO_Open R= bI_MANUAL_CMD;
	bClose_Cmd R= bDO_Close R= bI_MANUAL_CMD;
ELSE
	bOpen_Cmd R= bDO_Open R= NOT bI_MANUAL_CMD;
	bClose_Cmd R= bDO_Close R= NOT bI_MANUAL_CMD;
END_IF
bCmdActive := TRUE;
END_METHOD

END_FUNCTION_BLOCK

// Common/Measurement_Analog/fMeanFilter
FUNCTION fMeanFilter : REAL
VAR_INPUT
	rInputValue:REAL;
	rDelta:REAL;
END_VAR
VAR_IN_OUT
	rMeanValue:REAL;
END_VAR
VAR
END_VAR

rDelta := LIMIT(1,rDelta,100);
IF ABS(0.20*rMeanValue) < ABS( (rMeanValue - rInputValue)/rDelta) THEN
	rMeanValue := rInputValue;
END_IF
rMeanValue := rMeanValue - (rMeanValue - rInputValue)/rDelta;

END_FUNCTION

// Common/AlarmTable/fbAlarmSlaveTable
FUNCTION_BLOCK PUBLIC fbAlarmSlaveTable
VAR CONSTANT
	uiMaxRows:UINT := 20;
END_VAR
VAR_OUTPUT
	astErrTable			: ARRAY [1..20] OF stAlarmTableRow;		// Tabela z błędami
	uiRowNumber			: UINT;		// Aktualna liczba wierszy w tabeli
	uiRowsToRead		: UINT;		// Liczba nowych wierszy do odczytu przez bloczek nadrzędny
	bErrorOrUpActive	: BOOL:= FALSE;		// Aktywny alarm
	bWarningActive		: BOOL:= FALSE;		// Aktywne ostrzeżenie
	bInfoActive			: BOOL:= FALSE;		// Aktywna wiadomość
	dwLastErrorCode		: DWORD;			// Kod ostatniego błędu
END_VAR

ACTION aMesagesPoped:
uiRowsToRead := 0;
END_ACTION

METHOD mPushRow : BOOL
VAR_INPUT
	nAlarmClass:enAlarmClasses :=enAlarmClasses.Info;
	sMachineId:STRING(30);
	sEventDesc:STRING;
	dwErrorId:DWORD;
END_VAR
// Dodaj nowy alarm tylko gdy inny niż ostatni, jeśli taki sam zaktualizuj czas wystąpienia oraz zwiększ licznik wystąpień
IF sMachineId = astErrTable[1].sMachineId AND sEventDesc = astErrTable[1].sEventDescription THEN
	astErrTable[1].dtEventTime:= GVL_Aircom.stAC_DT_Data.dtActualDate;
	astErrTable[1].uiRepeatQty:= astErrTable[1].uiRepeatQty +1;
	uiRowsToRead := LIMIT(0,uiRowsToRead +1,uiMaxRows);
	IF nAlarmClass >= enAlarmClasses.Error THEN
		bErrorOrUpActive := TRUE;
		dwLastErrorCode := dwErrorId;
		bWarningActive := bInfoActive := FALSE;
	ELSIF nAlarmClass >= enAlarmClasses.Error THEN
		bWarningActive := TRUE;
		bInfoActive := FALSE;
	ELSIF nAlarmClass = enAlarmClasses.Info THEN
		bInfoActive := TRUE;
	END_IF
ELSE
	MEMMOVE (srcAddr := ADR(astErrTable[1]), destAddr := ADR(astErrTable[2]), n := ((uiMaxRows-1)*SIZEOF(astErrTable[1])) );
	astErrTable[1].dtEventTime:= GVL_Aircom.stAC_DT_Data.dtActualDate;
	astErrTable[1].sMachineId := sMachineId;
	astErrTable[1].sEventDescription := sEventDesc;
	astErrTable[1].dwErrorCode := dwErrorId;
	astErrTable[1].nAlarmClass := nAlarmClass;
	astErrTable[1].uiRepeatQty := 0;
	dwLastErrorCode := dwErrorId;
	bErrorOrUpActive S= nAlarmClass >= enAlarmClasses.Error;
	uiRowsToRead := LIMIT(0,uiRowsToRead +1,uiMaxRows);
	uiRowNumber := LIMIT(0,uiRowNumber +1,uiMaxRows);
END_IF
END_METHOD

METHOD mReset : BOOL
VAR_INPUT
END_VAR

VAR
END_VAR
MEMSET(destAddr := ADR(astErrTable), fillByte := 0, n := SIZEOF(astErrTable)); 
uiRowsToRead := uiRowNumber := 0;
bErrorOrUpActive := bInfoActive := bWarningActive := FALSE;
dwLastErrorCode := 0;
END_METHOD

END_FUNCTION_BLOCK

// Common/Actuator/fbActuatorOOP
FUNCTION_BLOCK fbActuatorOOP
VAR_IN_OUT
	stDigInOut: stActuatorDigInOut;
END_VAR
VAR_INPUT
	bI_Control_Ready:BOOL;					// Sygnał gotowości sterowania, sygnały otwórz/zamknij ustawiane tylko gdy jest gotowość
	bI_MANUAL_CMD:BOOL;						// Sygnał o ręcznym trybie sterowania
	bI_OpenInterlock:BOOL;					// Sygnał blokady otwierania zaworu/napędu (kolizja z innymi elementami) - powiązane z bI_RespectInterlockInMAN
	bI_CloseInterlock:BOOL;					// Sygnał blokady zamykania zaworu/napędu (kolizja z innymi elementami) - powiązane z bI_RespectInterlockInMAN
	bI_SusteinOpenPos:BOOL;					// Po dojściu do pozycji zadanej podtrzymaj sygnał sterujący - stosować np. dla zaworów 5/2 w celu podtrzymania zamknięcia
	bI_SusteinClosePos:BOOL;				// Po dojściu do pozycji zadanej podtrzymaj sygnał sterujący - stosować np. dla zaworów 5/2 w celu podtrzymania zamknięcia
	bI_RespectInterlockInMAN:BOOL:= TRUE;	// W trybie manualnym uwzględniaj interlocki czy nie
	bI_ResetErr:BOOL;
	bAllowOverCrossPosition:BOOL;			// Ustawiaj sygnał otwórz/zamknij gdy ustawi się odpowiednia krańcówka oraz gdy aktywny sygnał sterujący (zejście z krańcówki przy podtrzymaniu nie powoduje zaniku sygnału otwarcia/zamknięcia)
	bEnPossLossAlarm:BOOL:= FALSE;
	rI_OpenTime:REAL;
	rI_CloseTime:REAL;
	sActuatorId:STRING(30):= 'fbAct';
	sLangId:STRING(2);
	fbAlarmTab:REFERENCE TO fbAlarmSlaveTable;
END_VAR
VAR_OUTPUT
	bQ_Opened:BOOL;
	bQ_Closed:BOOL;
	bCmdActive:BOOL;
	bInMovement:BOOL;
END_VAR
VAR
	fbTON_OpenTimer:TON;
	fbTON_CloseTimer:TON;
	fbRTrig_Open:R_TRIG;
	fbRTrig_Close:R_TRIG;	
	fbRTrig_Ctr_Open:R_TRIG;
	fbRTrig_Ctr_Close:R_TRIG;	
	fbFTRIG_OpenPosition: F_TRIG;
	fbFTRIG_ClosePosition: F_TRIG;
	bOpen_Cmd: BOOL;
	bClose_Cmd: BOOL;
	fbFTrig_Opened: F_TRIG;
	fbFTrig_Closed: F_TRIG;
	rOpenMeanTime: REAL;
	rCloseMeanTime: REAL;
	bOpenTimeExceedAlSend: BOOL;
	bCloseTimeExceedAlSend: BOOL;
	bSwitchesErrorAlSend: BOOL;
	
	fbTON_controlReady: TON;
END_VAR

VAR PERSISTENT
	diNbOfOperations:DINT;
END_VAR


